LIN {X 0,Y 201.822,Z 772.403,A -85,B 0,C 180,E1 -21490.685,E2 -21490.685} C_VEL
LIN {X 0,Y 199.583,Z 777.598,A -85,B 0,C 180,E1 -21494.69,E2 -21494.69} C_VEL
LIN {X 0,Y 198.418,Z 780.58,A -85,B 0,C 180,E1 -21497.733,E2 -21497.733} C_VEL
LIN {X 0,Y 197.499,Z 783.514,A -85,B 0,C 180,E1 -21501.82,E2 -21501.82} C_VEL
LIN {X 0,Y 197.172,Z 785.274,A -85,B 0,C 180,E1 -21505.915,E2 -21505.915} C_VEL
LIN {X 0,Y 197.205,Z 785.884,A -85,B 0,C 180,E1 -21510.003,E2 -21510.003} C_VEL
LIN {X 0,Y 197.174,Z 785.308,A -85,B 0,C 180,E1 -21514.091,E2 -21514.091} C_VEL
LIN {X 0,Y 197.502,Z 783.592,A -85,B 0,C 180,E1 -21518.186,E2 -21518.186} C_VEL
LIN {X 0,Y 198.412,Z 780.698,A -85,B 0,C 180,E1 -21522.274,E2 -21522.274} C_VEL
LIN {X 0,Y 200.05,Z 776.56,A -85,B 0,C 180,E1 -21526.326,E2 -21526.326} C_VEL
LIN {X 0,Y 202.48,Z 770.918,A -85,B 0,C 180,E1 -21530.42,E2 -21530.42} C_VEL
LIN {X 0,Y 205.622,Z 764.102,A -85,B 0,C 180,E1 -21534.217,E2 -21534.217} C_VEL
LIN {X 0,Y 209.119,Z 756.621,A -85,B 0,C 180,E1 -21537.526,E2 -21537.526} C_VEL
LIN {X 0,Y 213.136,Z 748.003,A -85,B 0,C 180,E1 -21540.588,E2 -21540.588} C_VEL
LIN {X 0,Y 217.286,Z 738.403,A -85,B 0,C 180,E1 -21543.36,E2 -21543.36} C_VEL
LIN {X 0,Y 222.185,Z 726.543,A -85,B 0,C 180,E1 -21546.098,E2 -21546.098} C_VEL
LIN {X 0,Y 226.698,Z 714.44,A -85,B 0,C 180,E1 -21548.321,E2 -21548.321} C_VEL
LIN {X 0,Y 231.268,Z 700.736,A -85,B 0,C 180,E1 -21550.302,E2 -21550.302} C_VEL
LIN {X 0,Y 234.745,Z 688.105,A -85,B 0,C 180,E1 -21551.773,E2 -21551.773} C_VEL
LIN {X 0,Y 238.029,Z 673.847,A -85,B 0,C 180,E1 -21553.065,E2 -21553.065} C_VEL
LIN {X 0,Y 240.943,Z 658.425,A -85,B 0,C 180,E1 -21554.069,E2 -21554.069} C_VEL
LIN {X 0,Y 242.899,Z 642.997,A -85,B 0,C 180,E1 -21554.781,E2 -21554.781} C_VEL
LIN {X 0,Y 245.314,Z 607.777,A -85,B 0,C 180,E1 -21555.747,E2 -21555.747} C_VEL
LIN {X 0,Y 250.129,Z 529.748,A -85,B 0,C 180,E1 -21557.801,E2 -21557.801} C_VEL
LIN {X 0,Y 247.487,Z 500.103,A -85,B 0,C 180,E1 -21559.763,E2 -21559.763} C_VEL
LIN {X 0,Y 242.292,Z 488.929,A -85,B 0,C 180,E1 -21561.749,E2 -21561.749} C_VEL
LIN {X 0,Y 236.162,Z 477.144,A -85,B 0,C 180,E1 -21564.261,E2 -21564.261} C_VEL
LIN {X 0,Y 235.573,Z 475.998,A -85,B 0,C 180,E1 -21564.517,E2 -21564.517} C_VEL
LIN {X 0,Y 234.938,Z 476.527,A -85,B 0,C 180,E1 -21564.707,E2 -21564.707} C_VEL
LIN {X 0,Y 233.367,Z 478.417,A -85,B 0,C 180,E1 -21565.152,E2 -21565.152} C_VEL
LIN {X 0,Y 229.109,Z 492.899,A -85,B 0,C 180,E1 -21565.904,E2 -21565.904} C_VEL
LIN {X 0,Y 226.269,Z 500.58,A -85,B 0,C 180,E1 -21566.54,E2 -21566.54} C_VEL
LIN {X 0,Y 223.62,Z 505.401,A -85,B 0,C 180,E1 -21567.294,E2 -21567.294} C_VEL
LIN {X 0,Y 222.851,Z 506.93,A -85,B 0,C 180,E1 -21567.512,E2 -21567.512} C_VEL
LIN {X 0,Y 220.647,Z 514.522,A -85,B 0,C 180,E1 -21567.958,E2 -21567.958} C_VEL
LIN {X 0,Y 216.467,Z 529.632,A -85,B 0,C 180,E1 -21568.803,E2 -21568.803} C_VEL
LIN {X 0,Y 213.728,Z 537.354,A -85,B 0,C 180,E1 -21569.526,E2 -21569.526} C_VEL
LIN {X 0,Y 211.824,Z 540.819,A -85,B 0,C 180,E1 -21570.222,E2 -21570.222} C_VEL
LIN {X 0,Y 211.239,Z 542.496,A -85,B 0,C 180,E1 -21570.611,E2 -21570.611} C_VEL
LIN {X 0,Y 210.569,Z 548.908,A -85,B 0,C 180,E1 -21571.26,E2 -21571.26} C_VEL
LIN {X 0,Y 209.326,Z 568.525,A -85,B 0,C 180,E1 -21572.777,E2 -21572.777} C_VEL
LIN {X 0,Y 207.838,Z 584.724,A -85,B 0,C 180,E1 -21574.46,E2 -21574.46} C_VEL
LIN {X 0,Y 206.469,Z 599.243,A -85,B 0,C 180,E1 -21576.342,E2 -21576.342} C_VEL
LIN {X 0,Y 204.813,Z 613.408,A -85,B 0,C 180,E1 -21578.617,E2 -21578.617} C_VEL
LIN {X 0,Y 203.455,Z 626.182,A -85,B 0,C 180,E1 -21581.104,E2 -21581.104} C_VEL
LIN {X 0,Y 203.121,Z 628.887,A -85,B 0,C 180,E1 -21581.689,E2 -21581.689} C_VEL
LIN {X 0,Y 201.884,Z 633.396,A -85,B 0,C 180,E1 -21582.715,E2 -21582.715} C_VEL
LIN {X 0,Y 198.3,Z 640.449,A -85,B 0,C 180,E1 -21584.431,E2 -21584.431} C_VEL
LIN {X 0,Y 194.843,Z 647.157,A -85,B 0,C 180,E1 -21586.314,E2 -21586.314} C_VEL
LIN {X 0,Y 193.826,Z 651.128,A -85,B 0,C 180,E1 -21587.574,E2 -21587.574} C_VEL
LIN {X 0,Y 193.09,Z 661.092,A -85,B 0,C 180,E1 -21591.101,E2 -21591.101} C_VEL
LIN {X 0,Y 192.587,Z 669.692,A -85,B 0,C 180,E1 -21594.765,E2 -21594.765} C_VEL
LIN {X 0,Y 192.762,Z 677.727,A -85,B 0,C 180,E1 -21598.955,E2 -21598.955} C_VEL
LIN {X 0,Y 193.745,Z 684.126,A -85,B 0,C 180,E1 -21603.119,E2 -21603.119} C_VEL
LIN {X 0,Y 195.468,Z 689.048,A -85,B 0,C 180,E1 -21607.229,E2 -21607.229} C_VEL
LIN {X 0,Y 197.182,Z 691.828,A -85,B 0,C 180,E1 -21610.265,E2 -21610.265} C_VEL
LIN {X 0,Y 200.371,Z 694.455,A -85,B 0,C 180,E1 -21614.213,E2 -21614.213} C_VEL
LIN {X 0,Y 204.435,Z 695.846,A -85,B 0,C 180,E1 -21618.023,E2 -21618.023} C_VEL
LIN {X 0,Y 209.449,Z 696.032,A -85,B 0,C 180,E1 -21621.66,E2 -21621.66} C_VEL
LIN {X 0,Y 215.233,Z 695.074,A -85,B 0,C 180,E1 -21625.118,E2 -21625.118} C_VEL
LIN {X 0,Y 221.897,Z 692.933,A -85,B 0,C 180,E1 -21628.365,E2 -21628.365} C_VEL
LIN {X 0,Y 229.319,Z 689.599,A -85,B 0,C 180,E1 -21631.399,E2 -21631.399} C_VEL
LIN {X 0,Y 237.424,Z 685.083,A -85,B 0,C 180,E1 -21634.223,E2 -21634.223} C_VEL
LIN {X 0,Y 246.179,Z 679.309,A -85,B 0,C 180,E1 -21636.835,E2 -21636.835} C_VEL
LIN {X 0,Y 257.297,Z 670.804,A -85,B 0,C 180,E1 -21639.642,E2 -21639.642} C_VEL
LIN {X 0,Y 261.37,Z 667.332,A -85,B 0,C 180,E1 -21640.557,E2 -21640.557} C_VEL
LIN {X 0,Y 260.85,Z 668.132,A -85,B 0,C 180,E1 -21641.025,E2 -21641.025} C_VEL
LIN {X 0,Y 250.871,Z 678.551,A -85,B 0,C 180,E1 -21642.658,E2 -21642.658} C_VEL
LIN {X 0,Y 240.229,Z 688.929,A -85,B 0,C 180,E1 -21644.807,E2 -21644.807} C_VEL
LIN {X 0,Y 230.474,Z 697.908,A -85,B 0,C 180,E1 -21647.272,E2 -21647.272} C_VEL
LIN {X 0,Y 224.652,Z 703.275,A -85,B 0,C 180,E1 -21649.077,E2 -21649.077} C_VEL
LIN {X 0,Y 219.916,Z 716.568,A -85,B 0,C 180,E1 -21651.155,E2 -21651.155} C_VEL
LIN {X 0,Y 215.35,Z 728.239,A -85,B 0,C 180,E1 -21653.442,E2 -21653.442} C_VEL
LIN {X 0,Y 210.655,Z 738.922,A -85,B 0,C 180,E1 -21656.022,E2 -21656.022} C_VEL
LIN {X 0,Y 206.482,Z 748.241,A -85,B 0,C 180,E1 -21658.843,E2 -21658.843} C_VEL
LIN {X 0,Y 202.28,Z 756.832,A -85,B 0,C 180,E1 -21662.025,E2 -21662.025} C_VEL
LIN {X 0,Y 198.238,Z 765.11,A -85,B 0,C 180,E1 -21665.936,E2 -21665.936} C_VEL
LIN {X 0,Y 194.97,Z 771.854,A -85,B 0,C 180,E1 -21670.063,E2 -21670.063} C_VEL
LIN {X 0,Y 192.707,Z 776.915,A -85,B 0,C 180,E1 -21674.123,E2 -21674.123} C_VEL
LIN {X 0,Y 191.496,Z 779.895,A -85,B 0,C 180,E1 -21677.276,E2 -21677.276} C_VEL
LIN {X 0,Y 190.537,Z 782.809,A -85,B 0,C 180,E1 -21681.512,E2 -21681.512} C_VEL
LIN {X 0,Y 190.166,Z 784.542,A -85,B 0,C 180,E1 -21685.758,E2 -21685.758} C_VEL
LIN {X 0,Y 190.219,Z 785.129,A -85,B 0,C 180,E1 -21689.997,E2 -21689.997} C_VEL
LIN {X 0,Y 190.161,Z 784.528,A -85,B 0,C 180,E1 -21694.236,E2 -21694.236} C_VEL
LIN {X 0,Y 190.529,Z 782.778,A -85,B 0,C 180,E1 -21698.481,E2 -21698.481} C_VEL
LIN {X 0,Y 191.461,Z 779.852,A -85,B 0,C 180,E1 -21702.72,E2 -21702.72} C_VEL
LIN {X 0,Y 193.216,Z 775.677,A -85,B 0,C 180,E1 -21706.914,E2 -21706.914} C_VEL
LIN {X 0,Y 195.69,Z 770.141,A -85,B 0,C 180,E1 -21711.044,E2 -21711.044} C_VEL
LIN {X 0,Y 199.11,Z 763.093,A -85,B 0,C 180,E1 -21715.056,E2 -21715.056} C_VEL
LIN {X 0,Y 202.82,Z 755.539,A -85,B 0,C 180,E1 -21718.45,E2 -21718.45} C_VEL
LIN {X 0,Y 206.413,Z 748.128,A -85,B 0,C 180,E1 -21721.155,E2 -21721.155} C_VEL
LIN {X 0,Y 209.161,Z 741.992,A -85,B 0,C 180,E1 -21723.09,E2 -21723.09} C_VEL
LIN {X 0,Y 213.671,Z 731.872,A -85,B 0,C 180,E1 -21725.716,E2 -21725.716} C_VEL
LIN {X 0,Y 218.608,Z 719.81,A -85,B 0,C 180,E1 -21728.229,E2 -21728.229} C_VEL
LIN {X 0,Y 222.962,Z 707.693,A -85,B 0,C 180,E1 -21730.25,E2 -21730.25} C_VEL
LIN {X 0,Y 227.306,Z 693.77,A -85,B 0,C 180,E1 -21732.094,E2 -21732.094} C_VEL
LIN {X 0,Y 231.156,Z 678.884,A -85,B 0,C 180,E1 -21733.609,E2 -21733.609} C_VEL
LIN {X 0,Y 234.305,Z 663.775,A -85,B 0,C 180,E1 -21734.74,E2 -21734.74} C_VEL
LIN {X 0,Y 236.631,Z 648.765,A -85,B 0,C 180,E1 -21735.535,E2 -21735.535} C_VEL
LIN {X 0,Y 238.131,Z 633.231,A -85,B 0,C 180,E1 -21736.075,E2 -21736.075} C_VEL
LIN {X 0,Y 243.919,Z 543.137,A -85,B 0,C 180,E1 -21738.457,E2 -21738.457} C_VEL
LIN {X 0,Y 245.079,Z 524.954,A -85,B 0,C 180,E1 -21738.938,E2 -21738.938} C_VEL
LIN {X 0,Y 243.278,Z 494.459,A -85,B 0,C 180,E1 -21740.807,E2 -21740.807} C_VEL
LIN {X 0,Y 236.385,Z 475.168,A -85,B 0,C 180,E1 -21743.876,E2 -21743.876} C_VEL
LIN {X 0,Y 235.2,Z 472.841,A -85,B 0,C 180,E1 -21744.395,E2 -21744.395} C_VEL
LIN {X 0,Y 231.789,Z 467.9,A -85,B 0,C 180,E1 -21745.88,E2 -21745.88} C_VEL
LIN {X 0,Y 228.541,Z 461.545,A -85,B 0,C 180,E1 -21748.482,E2 -21748.482} C_VEL
LIN {X 0,Y 224.246,Z 454.408,A -85,B 0,C 180,E1 -21751.959,E2 -21751.959} C_VEL
LIN {X 0,Y 220.215,Z 447.535,A -85,B 0,C 180,E1 -21756.015,E2 -21756.015} C_VEL
LIN {X 0,Y 217.525,Z 443.267,A -85,B 0,C 180,E1 -21759.182,E2 -21759.182} C_VEL
LIN {X 0,Y 214.845,Z 439.385,A -85,B 0,C 180,E1 -21762.878,E2 -21762.878} C_VEL
LIN {X 0,Y 212.169,Z 434.902,A -85,B 0,C 180,E1 -21768.536,E2 -21768.536} C_VEL
LIN {X 0,Y 210.961,Z 433.332,A -85,B 0,C 180,E1 -21772.342,E2 -21772.342} C_VEL
LIN {X 0,Y 210.318,Z 432.552,A -85,B 0,C 180,E1 -21778.085,E2 -21778.085} C_VEL
LIN {X 0,Y 210.468,Z 432.967,A -85,B 0,C 180,E1 -21781.914,E2 -21781.914} C_VEL
LIN {X 0,Y 211.083,Z 434.259,A -85,B 0,C 180,E1 -21785.733,E2 -21785.733} C_VEL
LIN {X 0,Y 212.784,Z 438.249,A -85,B 0,C 180,E1 -21791.43,E2 -21791.43} C_VEL
LIN {X 0,Y 214.976,Z 442.904,A -85,B 0,C 180,E1 -21796.134,E2 -21796.134} C_VEL
LIN {X 0,Y 217.165,Z 447.743,A -85,B 0,C 180,E1 -21799.964,E2 -21799.964} C_VEL
LIN {X 0,Y 219.539,Z 453.313,A -85,B 0,C 180,E1 -21803.588,E2 -21803.588} C_VEL
LIN {X 0,Y 222.924,Z 461.584,A -85,B 0,C 180,E1 -21808.033,E2 -21808.033} C_VEL
LIN {X 0,Y 225.795,Z 469.875,A -85,B 0,C 180,E1 -21811.675,E2 -21811.675} C_VEL
LIN {X 0,Y 231.893,Z 480.479,A -85,B 0,C 180,E1 -21814.623,E2 -21814.623} C_VEL
LIN {X 0,Y 238.186,Z 492.808,A -85,B 0,C 180,E1 -21817.353,E2 -21817.353} C_VEL
LIN {X 0,Y 242.959,Z 503.436,A -85,B 0,C 180,E1 -21819.286,E2 -21819.286} C_VEL
LIN {X 0,Y 245.231,Z 531.174,A -85,B 0,C 180,E1 -21821.151,E2 -21821.151} C_VEL
LIN {X 0,Y 238.747,Z 630.862,A -85,B 0,C 180,E1 -21823.774,E2 -21823.774} C_VEL
LIN {X 0,Y 237.287,Z 647.272,A -85,B 0,C 180,E1 -21824.323,E2 -21824.323} C_VEL
LIN {X 0,Y 234.998,Z 662.794,A -85,B 0,C 180,E1 -21825.126,E2 -21825.126} C_VEL
LIN {X 0,Y 232.029,Z 677.096,A -85,B 0,C 180,E1 -21826.147,E2 -21826.147} C_VEL
LIN {X 0,Y 228.622,Z 690.646,A -85,B 0,C 180,E1 -21827.449,E2 -21827.449} C_VEL
LIN {X 0,Y 224.476,Z 704.619,A -85,B 0,C 180,E1 -21829.193,E2 -21829.193} C_VEL
LIN {X 0,Y 219.966,Z 717.307,A -85,B 0,C 180,E1 -21831.173,E2 -21831.173} C_VEL
LIN {X 0,Y 215.326,Z 728.928,A -85,B 0,C 180,E1 -21833.445,E2 -21833.445} C_VEL
LIN {X 0,Y 210.736,Z 739.581,A -85,B 0,C 180,E1 -21836.044,E2 -21836.044} C_VEL
LIN {X 0,Y 206.668,Z 748.771,A -85,B 0,C 180,E1 -21838.831,E2 -21838.831} C_VEL
LIN {X 0,Y 202.304,Z 757.469,A -85,B 0,C 180,E1 -21842.035,E2 -21842.035} C_VEL
LIN {X 0,Y 198.239,Z 765.746,A -85,B 0,C 180,E1 -21845.943,E2 -21845.943} C_VEL
LIN {X 0,Y 195.068,Z 772.389,A -85,B 0,C 180,E1 -21849.988,E2 -21849.988} C_VEL
LIN {X 0,Y 192.708,Z 777.584,A -85,B 0,C 180,E1 -21854.13,E2 -21854.13} C_VEL
LIN {X 0,Y 191.438,Z 780.566,A -85,B 0,C 180,E1 -21857.279,E2 -21857.279} C_VEL
LIN {X 0,Y 190.459,Z 783.5,A -85,B 0,C 180,E1 -21861.515,E2 -21861.515} C_VEL
LIN {X 0,Y 190.085,Z 785.261,A -85,B 0,C 180,E1 -21865.763,E2 -21865.763} C_VEL
LIN {X 0,Y 190.115,Z 785.87,A -85,B 0,C 180,E1 -21870.003,E2 -21870.003} C_VEL
LIN {X 0,Y 190.087,Z 785.294,A -85,B 0,C 180,E1 -21874.244,E2 -21874.244} C_VEL
LIN {X 0,Y 190.462,Z 783.577,A -85,B 0,C 180,E1 -21878.491,E2 -21878.491} C_VEL
LIN {X 0,Y 191.432,Z 780.683,A -85,B 0,C 180,E1 -21882.728,E2 -21882.728} C_VEL
LIN {X 0,Y 193.201,Z 776.544,A -85,B 0,C 180,E1 -21886.922,E2 -21886.922} C_VEL
LIN {X 0,Y 195.704,Z 771.063,A -85,B 0,C 180,E1 -21891.049,E2 -21891.049} C_VEL
LIN {X 0,Y 199.107,Z 764.084,A -85,B 0,C 180,E1 -21895.063,E2 -21895.063} C_VEL
LIN {X 0,Y 202.819,Z 756.602,A -85,B 0,C 180,E1 -21898.458,E2 -21898.458} C_VEL
LIN {X 0,Y 206.883,Z 748.24,A -85,B 0,C 180,E1 -21901.51,E2 -21901.51} C_VEL
LIN {X 0,Y 211.365,Z 738.381,A -85,B 0,C 180,E1 -21904.423,E2 -21904.423} C_VEL
LIN {X 0,Y 216.457,Z 726.518,A -85,B 0,C 180,E1 -21907.212,E2 -21907.212} C_VEL
LIN {X 0,Y 221.154,Z 714.412,A -85,B 0,C 180,E1 -21909.466,E2 -21909.466} C_VEL
LIN {X 0,Y 225.738,Z 701.182,A -85,B 0,C 180,E1 -21911.409,E2 -21911.409} C_VEL
LIN {X 0,Y 229.487,Z 688.066,A -85,B 0,C 180,E1 -21912.956,E2 -21912.956} C_VEL
LIN {X 0,Y 232.887,Z 673.799,A -85,B 0,C 180,E1 -21914.259,E2 -21914.259} C_VEL
LIN {X 0,Y 235.894,Z 658.359,A -85,B 0,C 180,E1 -21915.269,E2 -21915.269} C_VEL
LIN {X 0,Y 237.904,Z 642.891,A -85,B 0,C 180,E1 -21915.987,E2 -21915.987} C_VEL
LIN {X 0,Y 240.599,Z 605.269,A -85,B 0,C 180,E1 -21917.012,E2 -21917.012} C_VEL
LIN {X 0,Y 245.327,Z 530.521,A -85,B 0,C 180,E1 -21919.012,E2 -21919.012} C_VEL
LIN {X 0,Y 243.056,Z 503.406,A -85,B 0,C 180,E1 -21920.855,E2 -21920.855} C_VEL
LIN {X 0,Y 238.364,Z 493.238,A -85,B 0,C 180,E1 -21922.746,E2 -21922.746} C_VEL
LIN {X 0,Y 235.276,Z 487.003,A -85,B 0,C 180,E1 -21924.056,E2 -21924.056} C_VEL
LIN {X 0,Y 231.403,Z 499.009,A -85,B 0,C 180,E1 -21924.756,E2 -21924.756} C_VEL
LIN {X 0,Y 228.584,Z 505.786,A -85,B 0,C 180,E1 -21925.395,E2 -21925.395} C_VEL
LIN {X 0,Y 225.695,Z 510.994,A -85,B 0,C 180,E1 -21926.174,E2 -21926.174} C_VEL
LIN {X 0,Y 219.778,Z 531.993,A -85,B 0,C 180,E1 -21927.274,E2 -21927.274} C_VEL
LIN {X 0,Y 216.633,Z 540.683,A -85,B 0,C 180,E1 -21928.048,E2 -21928.048} C_VEL
LIN {X 0,Y 214.238,Z 545.202,A -85,B 0,C 180,E1 -21928.797,E2 -21928.797} C_VEL
LIN {X 0,Y 213.183,Z 546.946,A -85,B 0,C 180,E1 -21929.153,E2 -21929.153} C_VEL
LIN {X 0,Y 208.589,Z 562.229,A -85,B 0,C 180,E1 -21930.269,E2 -21930.269} C_VEL
LIN {X 0,Y 205.56,Z 570.357,A -85,B 0,C 180,E1 -21931.193,E2 -21931.193} C_VEL
LIN {X 0,Y 203.589,Z 574.003,A -85,B 0,C 180,E1 -21931.943,E2 -21931.943} C_VEL
LIN {X 0,Y 202.313,Z 575.787,A -85,B 0,C 180,E1 -21932.594,E2 -21932.594} C_VEL
LIN {X 0,Y 201.497,Z 579.228,A -85,B 0,C 180,E1 -21933.316,E2 -21933.316} C_VEL
LIN {X 0,Y 199.187,Z 601.55,A -85,B 0,C 180,E1 -21936.409,E2 -21936.409} C_VEL
LIN {X 0,Y 197.552,Z 615.998,A -85,B 0,C 180,E1 -21938.887,E2 -21938.887} C_VEL
LIN {X 0,Y 196.067,Z 628.546,A -85,B 0,C 180,E1 -21941.483,E2 -21941.483} C_VEL
LIN {X 0,Y 194.84,Z 639.997,A -85,B 0,C 180,E1 -21944.304,E2 -21944.304} C_VEL
LIN {X 0,Y 193.826,Z 651.128,A -85,B 0,C 180,E1 -21947.574,E2 -21947.574} C_VEL
LIN {X 0,Y 192.801,Z 655.036,A -85,B 0,C 180,E1 -21948.87,E2 -21948.87} C_VEL
LIN {X 0,Y 186.692,Z 665.347,A -85,B 0,C 180,E1 -21952.875,E2 -21952.875} C_VEL
LIN {X 0,Y 185.567,Z 668.609,A -85,B 0,C 180,E1 -21954.363,E2 -21954.363} C_VEL
LIN {X 0,Y 185.49,Z 669.682,A -85,B 0,C 180,E1 -21954.875,E2 -21954.875} C_VEL
LIN {X 0,Y 185.668,Z 677.422,A -85,B 0,C 180,E1 -21958.915,E2 -21958.915} C_VEL
LIN {X 0,Y 186.666,Z 684.138,A -85,B 0,C 180,E1 -21963.237,E2 -21963.237} C_VEL
LIN {X 0,Y 188.443,Z 689.389,A -85,B 0,C 180,E1 -21967.5,E2 -21967.5} C_VEL
LIN {X 0,Y 190.23,Z 692.476,A -85,B 0,C 180,E1 -21970.645,E2 -21970.645} C_VEL
LIN {X 0,Y 193.578,Z 695.43,A -85,B 0,C 180,E1 -21974.722,E2 -21974.722} C_VEL
LIN {X 0,Y 197.832,Z 697.169,A -85,B 0,C 180,E1 -21978.646,E2 -21978.646} C_VEL
LIN {X 0,Y 203.064,Z 697.7,A -85,B 0,C 180,E1 -21982.377,E2 -21982.377} C_VEL
LIN {X 0,Y 209.088,Z 697.103,A -85,B 0,C 180,E1 -21985.91,E2 -21985.91} C_VEL
LIN {X 0,Y 216.033,Z 695.352,A -85,B 0,C 180,E1 -21989.208,E2 -21989.208} C_VEL
LIN {X 0,Y 223.743,Z 692.456,A -85,B 0,C 180,E1 -21992.275,E2 -21992.275} C_VEL
LIN {X 0,Y 232.153,Z 688.406,A -85,B 0,C 180,E1 -21995.113,E2 -21995.113} C_VEL
LIN {X 0,Y 241.202,Z 683.173,A -85,B 0,C 180,E1 -21997.726,E2 -21997.726} C_VEL
LIN {X 0,Y 252,Z 675.891,A -85,B 0,C 180,E1 -22000.351,E2 -22000.351} C_VEL
LIN {X 0,Y 251.261,Z 676.688,A -85,B 0,C 180,E1 -22000.654,E2 -22000.654} C_VEL
LIN {X 0,Y 239.398,Z 687.495,A -85,B 0,C 180,E1 -22002.781,E2 -22002.781} C_VEL
LIN {X 0,Y 229.042,Z 696.348,A -85,B 0,C 180,E1 -22005.108,E2 -22005.108} C_VEL
LIN {X 0,Y 218.739,Z 704.998,A -85,B 0,C 180,E1 -22008.107,E2 -22008.107} C_VEL
LIN {X 0,Y 213.97,Z 717.756,A -85,B 0,C 180,E1 -22010.168,E2 -22010.168} C_VEL
LIN {X 0,Y 209.655,Z 728.263,A -85,B 0,C 180,E1 -22012.279,E2 -22012.279} C_VEL
LIN {X 0,Y 204.777,Z 738.944,A -85,B 0,C 180,E1 -22014.907,E2 -22014.907} C_VEL
LIN {X 0,Y 200.625,Z 747.724,A -85,B 0,C 180,E1 -22017.589,E2 -22017.589} C_VEL
LIN {X 0,Y 196.617,Z 755.678,A -85,B 0,C 180,E1 -22020.558,E2 -22020.558} C_VEL
LIN {X 0,Y 192.695,Z 763.212,A -85,B 0,C 180,E1 -22024.042,E2 -22024.042} C_VEL
LIN {X 0,Y 189.048,Z 770.233,A -85,B 0,C 180,E1 -22028.173,E2 -22028.173} C_VEL
LIN {X 0,Y 186.4,Z 775.746,A -85,B 0,C 180,E1 -22032.441,E2 -22032.441} C_VEL
LIN {X 0,Y 184.529,Z 779.91,A -85,B 0,C 180,E1 -22036.787,E2 -22036.787} C_VEL
LIN {X 0,Y 183.501,Z 782.823,A -85,B 0,C 180,E1 -22041.184,E2 -22041.184} C_VEL
LIN {X 0,Y 183.079,Z 784.556,A -85,B 0,C 180,E1 -22045.593,E2 -22045.593} C_VEL
LIN {X 0,Y 183.127,Z 785.142,A -85,B 0,C 180,E1 -22049.997,E2 -22049.997} C_VEL
LIN {X 0,Y 183.076,Z 784.542,A -85,B 0,C 180,E1 -22054.4,E2 -22054.4} C_VEL
LIN {X 0,Y 183.493,Z 782.792,A -85,B 0,C 180,E1 -22058.809,E2 -22058.809} C_VEL
LIN {X 0,Y 184.5,Z 779.865,A -85,B 0,C 180,E1 -22063.208,E2 -22063.208} C_VEL
LIN {X 0,Y 186.389,Z 775.691,A -85,B 0,C 180,E1 -22067.553,E2 -22067.553} C_VEL
LIN {X 0,Y 189.033,Z 770.155,A -85,B 0,C 180,E1 -22071.822,E2 -22071.822} C_VEL
LIN {X 0,Y 192.651,Z 763.107,A -85,B 0,C 180,E1 -22075.957,E2 -22075.957} C_VEL
LIN {X 0,Y 196.583,Z 755.554,A -85,B 0,C 180,E1 -22079.44,E2 -22079.44} C_VEL
LIN {X 0,Y 200.408,Z 747.899,A -85,B 0,C 180,E1 -22082.306,E2 -22082.306} C_VEL
LIN {X 0,Y 203.979,Z 740.396,A -85,B 0,C 180,E1 -22084.641,E2 -22084.641} C_VEL
LIN {X 0,Y 208.774,Z 730.004,A -85,B 0,C 180,E1 -22087.292,E2 -22087.292} C_VEL
LIN {X 0,Y 213.485,Z 718.691,A -85,B 0,C 180,E1 -22089.626,E2 -22089.626} C_VEL
LIN {X 0,Y 218.058,Z 706.38,A -85,B 0,C 180,E1 -22091.658,E2 -22091.658} C_VEL
LIN {X 0,Y 222.418,Z 692.669,A -85,B 0,C 180,E1 -22093.448,E2 -22093.448} C_VEL
LIN {X 0,Y 226.067,Z 678.917,A -85,B 0,C 180,E1 -22094.85,E2 -22094.85} C_VEL
LIN {X 0,Y 229.315,Z 663.818,A -85,B 0,C 180,E1 -22095.989,E2 -22095.989} C_VEL
LIN {X 0,Y 231.724,Z 648.828,A -85,B 0,C 180,E1 -22096.785,E2 -22096.785} C_VEL
LIN {X 0,Y 233.278,Z 633.332,A -85,B 0,C 180,E1 -22097.327,E2 -22097.327} C_VEL
LIN {X 0,Y 239.23,Z 544.075,A -85,B 0,C 180,E1 -22099.702,E2 -22099.702} C_VEL
LIN {X 0,Y 240.389,Z 524.977,A -85,B 0,C 180,E1 -22100.243,E2 -22100.243} C_VEL
LIN {X 0,Y 238.895,Z 497.387,A -85,B 0,C 180,E1 -22101.979,E2 -22101.979} C_VEL
LIN {X 0,Y 232.682,Z 479.464,A -85,B 0,C 180,E1 -22104.924,E2 -22104.924} C_VEL
LIN {X 0,Y 227.807,Z 472.074,A -85,B 0,C 180,E1 -22107.137,E2 -22107.137} C_VEL
LIN {X 0,Y 224.804,Z 467.654,A -85,B 0,C 180,E1 -22108.685,E2 -22108.685} C_VEL
LIN {X 0,Y 220.528,Z 460.091,A -85,B 0,C 180,E1 -22112.477,E2 -22112.477} C_VEL
LIN {X 0,Y 216.933,Z 453.901,A -85,B 0,C 180,E1 -22116.111,E2 -22116.111} C_VEL
LIN {X 0,Y 213.957,Z 449.133,A -85,B 0,C 180,E1 -22119.743,E2 -22119.743} C_VEL
LIN {X 0,Y 211.965,Z 446.122,A -85,B 0,C 180,E1 -22122.638,E2 -22122.638} C_VEL
LIN {X 0,Y 209.161,Z 441.496,A -85,B 0,C 180,E1 -22128.369,E2 -22128.369} C_VEL
LIN {X 0,Y 208.475,Z 440.425,A -85,B 0,C 180,E1 -22130.296,E2 -22130.296} C_VEL
LIN {X 0,Y 207.334,Z 439.366,A -85,B 0,C 180,E1 -22134.164,E2 -22134.164} C_VEL
LIN {X 0,Y 207.109,Z 438.88,A -85,B 0,C 180,E1 -22138.056,E2 -22138.056} C_VEL
LIN {X 0,Y 207.248,Z 439.318,A -85,B 0,C 180,E1 -22141.944,E2 -22141.944} C_VEL
LIN {X 0,Y 207.776,Z 440.659,A -85,B 0,C 180,E1 -22145.824,E2 -22145.824} C_VEL
LIN {X 0,Y 209.341,Z 444.672,A -85,B 0,C 180,E1 -22151.621,E2 -22151.621} C_VEL
LIN {X 0,Y 211.512,Z 449.47,A -85,B 0,C 180,E1 -22156.406,E2 -22156.406} C_VEL
LIN {X 0,Y 213.534,Z 454.252,A -85,B 0,C 180,E1 -22160.15,E2 -22160.15} C_VEL
LIN {X 0,Y 216.035,Z 460.411,A -85,B 0,C 180,E1 -22164.097,E2 -22164.097} C_VEL
LIN {X 0,Y 218.845,Z 467.738,A -85,B 0,C 180,E1 -22167.988,E2 -22167.988} C_VEL
LIN {X 0,Y 219.907,Z 470.403,A -85,B 0,C 180,E1 -22169.168,E2 -22169.168} C_VEL
LIN {X 0,Y 225.92,Z 480.721,A -85,B 0,C 180,E1 -22172.388,E2 -22172.388} C_VEL
LIN {X 0,Y 231.297,Z 490.851,A -85,B 0,C 180,E1 -22174.963,E2 -22174.963} C_VEL
LIN {X 0,Y 236,Z 500.733,A -85,B 0,C 180,E1 -22177.048,E2 -22177.048} C_VEL
LIN {X 0,Y 238.592,Z 506.663,A -85,B 0,C 180,E1 -22178.146,E2 -22178.146} C_VEL
LIN {X 0,Y 240.551,Z 532.006,A -85,B 0,C 180,E1 -22179.902,E2 -22179.902} C_VEL
LIN {X 0,Y 234.147,Z 627.191,A -85,B 0,C 180,E1 -22182.427,E2 -22182.427} C_VEL
LIN {X 0,Y 232.664,Z 645.062,A -85,B 0,C 180,E1 -22182.987,E2 -22182.987} C_VEL
LIN {X 0,Y 230.379,Z 660.554,A -85,B 0,C 180,E1 -22183.734,E2 -22183.734} C_VEL
LIN {X 0,Y 227.455,Z 674.873,A -85,B 0,C 180,E1 -22184.716,E2 -22184.716} C_VEL
LIN {X 0,Y 223.945,Z 688.894,A -85,B 0,C 180,E1 -22186.03,E2 -22186.03} C_VEL
LIN {X 0,Y 220.134,Z 701.678,A -85,B 0,C 180,E1 -22187.568,E2 -22187.568} C_VEL
LIN {X 0,Y 215.367,Z 714.979,A -85,B 0,C 180,E1 -22189.57,E2 -22189.57} C_VEL
LIN {X 0,Y 210.498,Z 726.987,A -85,B 0,C 180,E1 -22191.858,E2 -22191.858} C_VEL
LIN {X 0,Y 205.6,Z 737.956,A -85,B 0,C 180,E1 -22194.476,E2 -22194.476} C_VEL
LIN {X 0,Y 201.001,Z 747.846,A -85,B 0,C 180,E1 -22197.452,E2 -22197.452} C_VEL
LIN {X 0,Y 196.644,Z 756.272,A -85,B 0,C 180,E1 -22200.57,E2 -22200.57} C_VEL
LIN {X 0,Y 192.708,Z 763.807,A -85,B 0,C 180,E1 -22204.051,E2 -22204.051} C_VEL
LIN {X 0,Y 188.916,Z 771.231,A -85,B 0,C 180,E1 -22208.442,E2 -22208.442} C_VEL
LIN {X 0,Y 186.418,Z 776.376,A -85,B 0,C 180,E1 -22212.45,E2 -22212.45} C_VEL
LIN {X 0,Y 184.461,Z 780.553,A -85,B 0,C 180,E1 -22216.789,E2 -22216.789} C_VEL
LIN {X 0,Y 183.408,Z 783.486,A -85,B 0,C 180,E1 -22221.187,E2 -22221.187} C_VEL
LIN {X 0,Y 183.014,Z 785.247,A -85,B 0,C 180,E1 -22225.599,E2 -22225.599} C_VEL
LIN {X 0,Y 183.028,Z 785.856,A -85,B 0,C 180,E1 -22230.003,E2 -22230.003} C_VEL
LIN {X 0,Y 183.015,Z 785.28,A -85,B 0,C 180,E1 -22234.408,E2 -22234.408} C_VEL
LIN {X 0,Y 183.411,Z 783.563,A -85,B 0,C 180,E1 -22238.82,E2 -22238.82} C_VEL
LIN {X 0,Y 184.453,Z 780.668,A -85,B 0,C 180,E1 -22243.219,E2 -22243.219} C_VEL
LIN {X 0,Y 186.372,Z 776.529,A -85,B 0,C 180,E1 -22247.562,E2 -22247.562} C_VEL
LIN {X 0,Y 189.043,Z 771.046,A -85,B 0,C 180,E1 -22251.828,E2 -22251.828} C_VEL
LIN {X 0,Y 192.647,Z 764.066,A -85,B 0,C 180,E1 -22255.965,E2 -22255.965} C_VEL
LIN {X 0,Y 196.586,Z 756.583,A -85,B 0,C 180,E1 -22259.447,E2 -22259.447} C_VEL
LIN {X 0,Y 201.303,Z 747.153,A -85,B 0,C 180,E1 -22262.932,E2 -22262.932} C_VEL
LIN {X 0,Y 206.298,Z 736.664,A -85,B 0,C 180,E1 -22265.994,E2 -22265.994} C_VEL
LIN {X 0,Y 211.244,Z 725.454,A -85,B 0,C 180,E1 -22268.598,E2 -22268.598} C_VEL
LIN {X 0,Y 216.168,Z 713.135,A -85,B 0,C 180,E1 -22270.87,E2 -22270.87} C_VEL
LIN {X 0,Y 220.809,Z 699.918,A -85,B 0,C 180,E1 -22272.795,E2 -22272.795} C_VEL
LIN {X 0,Y 224.811,Z 686.156,A -85,B 0,C 180,E1 -22274.389,E2 -22274.389} C_VEL
LIN {X 0,Y 228.133,Z 672.581,A -85,B 0,C 180,E1 -22275.591,E2 -22275.591} C_VEL
LIN {X 0,Y 231.087,Z 657.44,A -85,B 0,C 180,E1 -22276.564,E2 -22276.564} C_VEL
LIN {X 0,Y 233.04,Z 642.784,A -85,B 0,C 180,E1 -22277.239,E2 -22277.239} C_VEL
LIN {X 0,Y 235.884,Z 604.057,A -85,B 0,C 180,E1 -22278.303,E2 -22278.303} C_VEL
LIN {X 0,Y 240.66,Z 532.179,A -85,B 0,C 180,E1 -22280.225,E2 -22280.225} C_VEL
LIN {X 0,Y 238.7,Z 506.724,A -85,B 0,C 180,E1 -22281.991,E2 -22281.991} C_VEL
LIN {X 0,Y 235.792,Z 500.201,A -85,B 0,C 180,E1 -22283.223,E2 -22283.223} C_VEL
LIN {X 0,Y 235.566,Z 500.122,A -85,B 0,C 180,E1 -22283.3,E2 -22283.3} C_VEL
LIN {X 0,Y 232.248,Z 508.399,A -85,B 0,C 180,E1 -22283.978,E2 -22283.978} C_VEL
LIN {X 0,Y 228.799,Z 514.787,A -85,B 0,C 180,E1 -22284.835,E2 -22284.835} C_VEL
LIN {X 0,Y 223.521,Z 533.48,A -85,B 0,C 180,E1 -22285.735,E2 -22285.735} C_VEL
LIN {X 0,Y 219.939,Z 543.423,A -85,B 0,C 180,E1 -22286.541,E2 -22286.541} C_VEL
LIN {X 0,Y 217.317,Z 548.651,A -85,B 0,C 180,E1 -22287.282,E2 -22287.282} C_VEL
LIN {X 0,Y 215.749,Z 551.434,A -85,B 0,C 180,E1 -22287.763,E2 -22287.763} C_VEL
LIN {X 0,Y 211.778,Z 564.569,A -85,B 0,C 180,E1 -22288.651,E2 -22288.651} C_VEL
LIN {X 0,Y 208.233,Z 573.872,A -85,B 0,C 180,E1 -22289.655,E2 -22289.655} C_VEL
LIN {X 0,Y 205.624,Z 578.752,A -85,B 0,C 180,E1 -22290.572,E2 -22290.572} C_VEL
LIN {X 0,Y 203.227,Z 582.177,A -85,B 0,C 180,E1 -22291.537,E2 -22291.537} C_VEL
LIN {X 0,Y 197.585,Z 596.555,A -85,B 0,C 180,E1 -22293.53,E2 -22293.53} C_VEL
LIN {X 0,Y 194.496,Z 602.76,A -85,B 0,C 180,E1 -22294.876,E2 -22294.876} C_VEL
LIN {X 0,Y 192.614,Z 605.229,A -85,B 0,C 180,E1 -22295.908,E2 -22295.908} C_VEL
LIN {X 0,Y 191.938,Z 606.321,A -85,B 0,C 180,E1 -22296.482,E2 -22296.482} C_VEL
LIN {X 0,Y 191.027,Z 610.771,A -85,B 0,C 180,E1 -22297.632,E2 -22297.632} C_VEL
LIN {X 0,Y 189.331,Z 625.927,A -85,B 0,C 180,E1 -22300.765,E2 -22300.765} C_VEL
LIN {X 0,Y 187.912,Z 638.083,A -85,B 0,C 180,E1 -22303.71,E2 -22303.71} C_VEL
LIN {X 0,Y 186.904,Z 649.205,A -85,B 0,C 180,E1 -22306.961,E2 -22306.961} C_VEL
LIN {X 0,Y 186.06,Z 660.07,A -85,B 0,C 180,E1 -22310.762,E2 -22310.762} C_VEL
LIN {X 0,Y 185.484,Z 669.037,A -85,B 0,C 180,E1 -22314.564,E2 -22314.564} C_VEL
LIN {X 0,Y 185.49,Z 669.682,A -85,B 0,C 180,E1 -22314.875,E2 -22314.875} C_VEL
LIN {X 0,Y 184.885,Z 672.807,A -85,B 0,C 180,E1 -22316.414,E2 -22316.414} C_VEL
LIN {X 0,Y 182.235,Z 677.532,A -85,B 0,C 180,E1 -22319,E2 -22319} C_VEL
LIN {X 0,Y 179.815,Z 681.818,A -85,B 0,C 180,E1 -22321.737,E2 -22321.737} C_VEL
LIN {X 0,Y 179.595,Z 684.222,A -85,B 0,C 180,E1 -22323.463,E2 -22323.463} C_VEL
LIN {X 0,Y 181.427,Z 689.679,A -85,B 0,C 180,E1 -22327.792,E2 -22327.792} C_VEL
LIN {X 0,Y 183.283,Z 692.951,A -85,B 0,C 180,E1 -22331.053,E2 -22331.053} C_VEL
LIN {X 0,Y 186.765,Z 696.244,A -85,B 0,C 180,E1 -22335.272,E2 -22335.272} C_VEL
LIN {X 0,Y 191.211,Z 698.336,A -85,B 0,C 180,E1 -22339.317,E2 -22339.317} C_VEL
LIN {X 0,Y 196.689,Z 699.244,A -85,B 0,C 180,E1 -22343.144,E2 -22343.144} C_VEL
LIN {X 0,Y 202.967,Z 699.048,A -85,B 0,C 180,E1 -22346.753,E2 -22346.753} C_VEL
LIN {X 0,Y 210.205,Z 697.711,A -85,B 0,C 180,E1 -22350.1,E2 -22350.1} C_VEL
LIN {X 0,Y 218.213,Z 695.261,A -85,B 0,C 180,E1 -22353.197,E2 -22353.197} C_VEL
LIN {X 0,Y 226.907,Z 691.685,A -85,B 0,C 180,E1 -22356.049,E2 -22356.049} C_VEL
LIN {X 0,Y 236.284,Z 686.953,A -85,B 0,C 180,E1 -22358.654,E2 -22358.654} C_VEL
LIN {X 0,Y 241.223,Z 684.131,A -85,B 0,C 180,E1 -22359.864,E2 -22359.864} C_VEL
LIN {X 0,Y 241.384,Z 684.28,A -85,B 0,C 180,E1 -22360.341,E2 -22360.341} C_VEL
LIN {X 0,Y 229.351,Z 693.906,A -85,B 0,C 180,E1 -22362.653,E2 -22362.653} C_VEL
LIN {X 0,Y 219.212,Z 701.537,A -85,B 0,C 180,E1 -22365.141,E2 -22365.141} C_VEL
LIN {X 0,Y 213.017,Z 706.39,A -85,B 0,C 180,E1 -22367.035,E2 -22367.035} C_VEL
LIN {X 0,Y 208.084,Z 718.945,A -85,B 0,C 180,E1 -22369.124,E2 -22369.124} C_VEL
LIN {X 0,Y 203.216,Z 730.221,A -85,B 0,C 180,E1 -22371.497,E2 -22371.497} C_VEL
LIN {X 0,Y 198.166,Z 740.58,A -85,B 0,C 180,E1 -22374.181,E2 -22374.181} C_VEL
LIN {X 0,Y 193.827,Z 749.352,A -85,B 0,C 180,E1 -22377.048,E2 -22377.048} C_VEL
LIN {X 0,Y 189.145,Z 757.977,A -85,B 0,C 180,E1 -22380.503,E2 -22380.503} C_VEL
LIN {X 0,Y 185.264,Z 765.144,A -85,B 0,C 180,E1 -22384.132,E2 -22384.132} C_VEL
LIN {X 0,Y 181.853,Z 771.286,A -85,B 0,C 180,E1 -22388.05,E2 -22388.05} C_VEL
LIN {X 0,Y 178.994,Z 776.946,A -85,B 0,C 180,E1 -22392.87,E2 -22392.87} C_VEL
LIN {X 0,Y 177.563,Z 779.925,A -85,B 0,C 180,E1 -22396.259,E2 -22396.259} C_VEL
LIN {X 0,Y 176.455,Z 782.838,A -85,B 0,C 180,E1 -22400.829,E2 -22400.829} C_VEL
LIN {X 0,Y 176.008,Z 784.57,A -85,B 0,C 180,E1 -22405.416,E2 -22405.416} C_VEL
LIN {X 0,Y 176.037,Z 785.156,A -85,B 0,C 180,E1 -22409.996,E2 -22409.996} C_VEL
LIN {X 0,Y 176.006,Z 784.556,A -85,B 0,C 180,E1 -22414.577,E2 -22414.577} C_VEL
LIN {X 0,Y 176.447,Z 782.806,A -85,B 0,C 180,E1 -22419.164,E2 -22419.164} C_VEL
LIN {X 0,Y 177.536,Z 779.879,A -85,B 0,C 180,E1 -22423.736,E2 -22423.736} C_VEL
LIN {X 0,Y 179.567,Z 775.705,A -85,B 0,C 180,E1 -22428.243,E2 -22428.243} C_VEL
LIN {X 0,Y 182.406,Z 770.169,A -85,B 0,C 180,E1 -22432.658,E2 -22432.658} C_VEL
LIN {X 0,Y 186.26,Z 763.122,A -85,B 0,C 180,E1 -22436.918,E2 -22436.918} C_VEL
LIN {X 0,Y 190.411,Z 755.569,A -85,B 0,C 180,E1 -22440.494,E2 -22440.494} C_VEL
LIN {X 0,Y 194.258,Z 748.17,A -85,B 0,C 180,E1 -22443.343,E2 -22443.343} C_VEL
LIN {X 0,Y 198.138,Z 740.413,A -85,B 0,C 180,E1 -22445.817,E2 -22445.817} C_VEL
LIN {X 0,Y 203.144,Z 730.022,A -85,B 0,C 180,E1 -22448.511,E2 -22448.511} C_VEL
LIN {X 0,Y 208.055,Z 718.711,A -85,B 0,C 180,E1 -22450.875,E2 -22450.875} C_VEL
LIN {X 0,Y 212.798,Z 706.402,A -85,B 0,C 180,E1 -22452.931,E2 -22452.931} C_VEL
LIN {X 0,Y 217.125,Z 693.364,A -85,B 0,C 180,E1 -22454.66,E2 -22454.66} C_VEL
LIN {X 0,Y 221.094,Z 678.949,A -85,B 0,C 180,E1 -22456.147,E2 -22456.147} C_VEL
LIN {X 0,Y 224.454,Z 663.86,A -85,B 0,C 180,E1 -22457.289,E2 -22457.289} C_VEL
LIN {X 0,Y 226.932,Z 648.889,A -85,B 0,C 180,E1 -22458.089,E2 -22458.089} C_VEL
LIN {X 0,Y 228.539,Z 633.431,A -85,B 0,C 180,E1 -22458.632,E2 -22458.632} C_VEL
LIN {X 0,Y 234.76,Z 543.311,A -85,B 0,C 180,E1 -22461.048,E2 -22461.048} C_VEL
LIN {X 0,Y 235.864,Z 526.059,A -85,B 0,C 180,E1 -22461.536,E2 -22461.536} C_VEL
LIN {X 0,Y 234.618,Z 500.314,A -85,B 0,C 180,E1 -22463.195,E2 -22463.195} C_VEL
LIN {X 0,Y 229.22,Z 484.16,A -85,B 0,C 180,E1 -22465.923,E2 -22465.923} C_VEL
LIN {X 0,Y 222.035,Z 473.504,A -85,B 0,C 180,E1 -22469.442,E2 -22469.442} C_VEL
LIN {X 0,Y 217.838,Z 467.78,A -85,B 0,C 180,E1 -22471.846,E2 -22471.846} C_VEL
LIN {X 0,Y 214.044,Z 461.086,A -85,B 0,C 180,E1 -22475.768,E2 -22475.768} C_VEL
LIN {X 0,Y 210.984,Z 455.871,A -85,B 0,C 180,E1 -22479.527,E2 -22479.527} C_VEL
LIN {X 0,Y 207.847,Z 451.149,A -85,B 0,C 180,E1 -22484.306,E2 -22484.306} C_VEL
LIN {X 0,Y 206.147,Z 448.082,A -85,B 0,C 180,E1 -22488.197,E2 -22488.197} C_VEL
LIN {X 0,Y 205.479,Z 446.955,A -85,B 0,C 180,E1 -22490.153,E2 -22490.153} C_VEL
LIN {X 0,Y 204.871,Z 446.193,A -85,B 0,C 180,E1 -22492.113,E2 -22492.113} C_VEL
LIN {X 0,Y 203.905,Z 445.199,A -85,B 0,C 180,E1 -22498.147,E2 -22498.147} C_VEL
LIN {X 0,Y 204.034,Z 445.656,A -85,B 0,C 180,E1 -22501.974,E2 -22501.974} C_VEL
LIN {X 0,Y 204.54,Z 447.071,A -85,B 0,C 180,E1 -22505.917,E2 -22505.917} C_VEL
LIN {X 0,Y 206.006,Z 451.201,A -85,B 0,C 180,E1 -22511.812,E2 -22511.812} C_VEL
LIN {X 0,Y 208.044,Z 456.043,A -85,B 0,C 180,E1 -22516.687,E2 -22516.687} C_VEL
LIN {X 0,Y 210,Z 460.953,A -85,B 0,C 180,E1 -22520.446,E2 -22520.446} C_VEL
LIN {X 0,Y 211.862,Z 465.675,A -85,B 0,C 180,E1 -22523.458,E2 -22523.458} C_VEL
LIN {X 0,Y 213.605,Z 470.187,A -85,B 0,C 180,E1 -22525.977,E2 -22525.977} C_VEL
LIN {X 0,Y 218.427,Z 478.171,A -85,B 0,C 180,E1 -22528.989,E2 -22528.989} C_VEL
LIN {X 0,Y 223.698,Z 487.608,A -85,B 0,C 180,E1 -22531.895,E2 -22531.895} C_VEL
LIN {X 0,Y 228.895,Z 497.846,A -85,B 0,C 180,E1 -22534.478,E2 -22534.478} C_VEL
LIN {X 0,Y 233.309,Z 507.607,A -85,B 0,C 180,E1 -22536.517,E2 -22536.517} C_VEL
LIN {X 0,Y 234.371,Z 510.608,A -85,B 0,C 180,E1 -22537.014,E2 -22537.014} C_VEL
LIN {X 0,Y 235.983,Z 533.03,A -85,B 0,C 180,E1 -22538.611,E2 -22538.611} C_VEL
LIN {X 0,Y 229.412,Z 627.09,A -85,B 0,C 180,E1 -22541.117,E2 -22541.117} C_VEL
LIN {X 0,Y 227.892,Z 644.999,A -85,B 0,C 180,E1 -22541.684,E2 -22541.684} C_VEL
LIN {X 0,Y 225.525,Z 660.511,A -85,B 0,C 180,E1 -22542.429,E2 -22542.429} C_VEL
LIN {X 0,Y 222.518,Z 674.84,A -85,B 0,C 180,E1 -22543.417,E2 -22543.417} C_VEL
LIN {X 0,Y 218.887,Z 688.867,A -85,B 0,C 180,E1 -22544.738,E2 -22544.738} C_VEL
LIN {X 0,Y 214.846,Z 701.871,A -85,B 0,C 180,E1 -22546.315,E2 -22546.315} C_VEL
LIN {X 0,Y 210.002,Z 714.958,A -85,B 0,C 180,E1 -22548.311,E2 -22548.311} C_VEL
LIN {X 0,Y 204.922,Z 726.968,A -85,B 0,C 180,E1 -22550.623,E2 -22550.623} C_VEL
LIN {X 0,Y 199.832,Z 737.939,A -85,B 0,C 180,E1 -22553.286,E2 -22553.286} C_VEL
LIN {X 0,Y 195.458,Z 746.73,A -85,B 0,C 180,E1 -22555.942,E2 -22555.942} C_VEL
LIN {X 0,Y 191.164,Z 755.04,A -85,B 0,C 180,E1 -22559.027,E2 -22559.027} C_VEL
LIN {X 0,Y 187.406,Z 761.797,A -85,B 0,C 180,E1 -22562.05,E2 -22562.05} C_VEL
LIN {X 0,Y 183.345,Z 769.23,A -85,B 0,C 180,E1 -22566.27,E2 -22566.27} C_VEL
LIN {X 0,Y 180.211,Z 775.131,A -85,B 0,C 180,E1 -22570.645,E2 -22570.645} C_VEL
LIN {X 0,Y 178.434,Z 778.612,A -85,B 0,C 180,E1 -22574,E2 -22574} C_VEL
LIN {X 0,Y 176.86,Z 782.156,A -85,B 0,C 180,E1 -22578.543,E2 -22578.543} C_VEL
LIN {X 0,Y 176.072,Z 784.497,A -85,B 0,C 180,E1 -22583.126,E2 -22583.126} C_VEL
LIN {X 0,Y 175.887,Z 785.685,A -85,B 0,C 180,E1 -22587.714,E2 -22587.714} C_VEL
LIN {X 0,Y 175.937,Z 785.842,A -85,B 0,C 180,E1 -22590.004,E2 -22590.004} C_VEL
LIN {X 0,Y 175.937,Z 785.266,A -85,B 0,C 180,E1 -22594.586,E2 -22594.586} C_VEL
LIN {X 0,Y 176.357,Z 783.548,A -85,B 0,C 180,E1 -22599.176,E2 -22599.176} C_VEL
LIN {X 0,Y 177.492,Z 780.653,A -85,B 0,C 180,E1 -22603.747,E2 -22603.747} C_VEL
LIN {X 0,Y 179.551,Z 776.513,A -85,B 0,C 180,E1 -22608.252,E2 -22608.252} C_VEL
LIN {X 0,Y 182.415,Z 771.029,A -85,B 0,C 180,E1 -22612.664,E2 -22612.664} C_VEL
LIN {X 0,Y 186.244,Z 764.048,A -85,B 0,C 180,E1 -22616.928,E2 -22616.928} C_VEL
LIN {X 0,Y 190.413,Z 756.564,A -85,B 0,C 180,E1 -22620.501,E2 -22620.501} C_VEL
LIN {X 0,Y 195.041,Z 747.73,A -85,B 0,C 180,E1 -22623.877,E2 -22623.877} C_VEL
LIN {X 0,Y 199.744,Z 738.337,A -85,B 0,C 180,E1 -22626.74,E2 -22626.74} C_VEL
LIN {X 0,Y 205.272,Z 726.468,A -85,B 0,C 180,E1 -22629.622,E2 -22629.622} C_VEL
LIN {X 0,Y 210.359,Z 714.355,A -85,B 0,C 180,E1 -22631.931,E2 -22631.931} C_VEL
LIN {X 0,Y 215.369,Z 700.737,A -85,B 0,C 180,E1 -22633.971,E2 -22633.971} C_VEL
LIN {X 0,Y 219.276,Z 687.989,A -85,B 0,C 180,E1 -22635.494,E2 -22635.494} C_VEL
LIN {X 0,Y 222.954,Z 673.704,A -85,B 0,C 180,E1 -22636.802,E2 -22636.802} C_VEL
LIN {X 0,Y 226.129,Z 658.224,A -85,B 0,C 180,E1 -22637.825,E2 -22637.825} C_VEL
LIN {X 0,Y 228.288,Z 642.674,A -85,B 0,C 180,E1 -22638.545,E2 -22638.545} C_VEL
LIN {X 0,Y 231.375,Z 601.832,A -85,B 0,C 180,E1 -22639.67,E2 -22639.67} C_VEL
LIN {X 0,Y 236.079,Z 532.786,A -85,B 0,C 180,E1 -22641.543,E2 -22641.543} C_VEL
LIN {X 0,Y 234.712,Z 513.636,A -85,B 0,C 180,E1 -22642.903,E2 -22642.903} C_VEL
LIN {X 0,Y 232.224,Z 518.14,A -85,B 0,C 180,E1 -22643.488,E2 -22643.488} C_VEL
LIN {X 0,Y 227.045,Z 536.113,A -85,B 0,C 180,E1 -22644.318,E2 -22644.318} C_VEL
LIN {X 0,Y 223.137,Z 546.732,A -85,B 0,C 180,E1 -22645.143,E2 -22645.143} C_VEL
LIN {X 0,Y 220.154,Z 552.683,A -85,B 0,C 180,E1 -22645.927,E2 -22645.927} C_VEL
LIN {X 0,Y 218.758,Z 555.05,A -85,B 0,C 180,E1 -22646.331,E2 -22646.331} C_VEL
LIN {X 0,Y 215.132,Z 566.893,A -85,B 0,C 180,E1 -22647.083,E2 -22647.083} C_VEL
LIN {X 0,Y 211.2,Z 577.097,A -85,B 0,C 180,E1 -22648.112,E2 -22648.112} C_VEL
LIN {X 0,Y 208.187,Z 582.886,A -85,B 0,C 180,E1 -22649.08,E2 -22649.08} C_VEL
LIN {X 0,Y 205.139,Z 587.369,A -85,B 0,C 180,E1 -22650.214,E2 -22650.214} C_VEL
LIN {X 0,Y 200.166,Z 599.812,A -85,B 0,C 180,E1 -22651.848,E2 -22651.848} C_VEL
LIN {X 0,Y 196.5,Z 607.159,A -85,B 0,C 180,E1 -22653.314,E2 -22653.314} C_VEL
LIN {X 0,Y 194.285,Z 610.352,A -85,B 0,C 180,E1 -22654.367,E2 -22654.367} C_VEL
LIN {X 0,Y 192.499,Z 612.331,A -85,B 0,C 180,E1 -22655.318,E2 -22655.318} C_VEL
LIN {X 0,Y 186.488,Z 625.463,A -85,B 0,C 180,E1 -22658.297,E2 -22658.297} C_VEL
LIN {X 0,Y 183.527,Z 630.744,A -85,B 0,C 180,E1 -22660.131,E2 -22660.131} C_VEL
LIN {X 0,Y 182.205,Z 632.403,A -85,B 0,C 180,E1 -22661.153,E2 -22661.153} C_VEL
LIN {X 0,Y 181.549,Z 633.474,A -85,B 0,C 180,E1 -22661.959,E2 -22661.959} C_VEL
LIN {X 0,Y 180.915,Z 637.21,A -85,B 0,C 180,E1 -22663.351,E2 -22663.351} C_VEL
LIN {X 0,Y 179.642,Z 650.993,A -85,B 0,C 180,E1 -22667.575,E2 -22667.575} C_VEL
LIN {X 0,Y 178.786,Z 661.709,A -85,B 0,C 180,E1 -22671.523,E2 -22671.523} C_VEL
LIN {X 0,Y 178.419,Z 670.59,A -85,B 0,C 180,E1 -22675.481,E2 -22675.481} C_VEL
LIN {X 0,Y 178.579,Z 676.984,A -85,B 0,C 180,E1 -22678.872,E2 -22678.872} C_VEL
LIN {X 0,Y 179.595,Z 684.222,A -85,B 0,C 180,E1 -22683.463,E2 -22683.463} C_VEL
LIN {X 0,Y 179.518,Z 686.533,A -85,B 0,C 180,E1 -22685.205,E2 -22685.205} C_VEL
LIN {X 0,Y 177.938,Z 689.968,A -85,B 0,C 180,E1 -22688.145,E2 -22688.145} C_VEL
LIN {X 0,Y 176.873,Z 692.452,A -85,B 0,C 180,E1 -22690.563,E2 -22690.563} C_VEL
LIN {X 0,Y 177.066,Z 694.185,A -85,B 0,C 180,E1 -22692.397,E2 -22692.397} C_VEL
LIN {X 0,Y 177.431,Z 694.715,A -85,B 0,C 180,E1 -22692.999,E2 -22692.999} C_VEL
LIN {X 0,Y 179.973,Z 697.013,A -85,B 0,C 180,E1 -22695.864,E2 -22695.864} C_VEL
LIN {X 0,Y 184.615,Z 699.449,A -85,B 0,C 180,E1 -22700.036,E2 -22700.036} C_VEL
LIN {X 0,Y 190.332,Z 700.707,A -85,B 0,C 180,E1 -22703.964,E2 -22703.964} C_VEL
LIN {X 0,Y 196.869,Z 700.876,A -85,B 0,C 180,E1 -22707.651,E2 -22707.651} C_VEL
LIN {X 0,Y 204.4,Z 699.922,A -85,B 0,C 180,E1 -22711.048,E2 -22711.048} C_VEL
LIN {X 0,Y 212.692,Z 697.903,A -85,B 0,C 180,E1 -22714.175,E2 -22714.175} C_VEL
LIN {X 0,Y 221.688,Z 694.799,A -85,B 0,C 180,E1 -22717.037,E2 -22717.037} C_VEL
LIN {X 0,Y 231.363,Z 690.589,A -85,B 0,C 180,E1 -22719.636,E2 -22719.636} C_VEL
LIN {X 0,Y 230.224,Z 691.657,A -85,B 0,C 180,E1 -22720.252,E2 -22720.252} C_VEL
LIN {X 0,Y 219.397,Z 699.228,A -85,B 0,C 180,E1 -22722.54,E2 -22722.54} C_VEL
LIN {X 0,Y 207.48,Z 707.443,A -85,B 0,C 180,E1 -22725.848,E2 -22725.848} C_VEL
LIN {X 0,Y 202.28,Z 720.091,A -85,B 0,C 180,E1 -22728.02,E2 -22728.02} C_VEL
LIN {X 0,Y 196.791,Z 732.113,A -85,B 0,C 180,E1 -22730.658,E2 -22730.658} C_VEL
LIN {X 0,Y 191.614,Z 742.206,A -85,B 0,C 180,E1 -22733.411,E2 -22733.411} C_VEL
LIN {X 0,Y 186.446,Z 752.045,A -85,B 0,C 180,E1 -22736.864,E2 -22736.864} C_VEL
LIN {X 0,Y 181.712,Z 760.213,A -85,B 0,C 180,E1 -22740.45,E2 -22740.45} C_VEL
LIN {X 0,Y 177.773,Z 766.957,A -85,B 0,C 180,E1 -22744.22,E2 -22744.22} C_VEL
LIN {X 0,Y 174.198,Z 773.199,A -85,B 0,C 180,E1 -22748.706,E2 -22748.706} C_VEL
LIN {X 0,Y 171.593,Z 778.02,A -85,B 0,C 180,E1 -22753.336,E2 -22753.336} C_VEL
LIN {X 0,Y 169.941,Z 781.548,A -85,B 0,C 180,E1 -22758.063,E2 -22758.063} C_VEL
LIN {X 0,Y 169.096,Z 783.862,A -85,B 0,C 180,E1 -22762.834,E2 -22762.834} C_VEL
LIN {X 0,Y 168.887,Z 785.02,A -85,B 0,C 180,E1 -22767.611,E2 -22767.611} C_VEL
LIN {X 0,Y 168.949,Z 785.17,A -85,B 0,C 180,E1 -22769.996,E2 -22769.996} C_VEL
LIN {X 0,Y 168.929,Z 784.569,A -85,B 0,C 180,E1 -22774.769,E2 -22774.769} C_VEL
LIN {X 0,Y 169.398,Z 782.819,A -85,B 0,C 180,E1 -22779.549,E2 -22779.549} C_VEL
LIN {X 0,Y 170.592,Z 779.893,A -85,B 0,C 180,E1 -22784.307,E2 -22784.307} C_VEL
LIN {X 0,Y 172.762,Z 775.719,A -85,B 0,C 180,E1 -22788.988,E2 -22788.988} C_VEL
LIN {X 0,Y 175.815,Z 770.183,A -85,B 0,C 180,E1 -22793.558,E2 -22793.558} C_VEL
LIN {X 0,Y 179.899,Z 763.137,A -85,B 0,C 180,E1 -22797.952,E2 -22797.952} C_VEL
LIN {X 0,Y 184.303,Z 755.584,A -85,B 0,C 180,E1 -22801.619,E2 -22801.619} C_VEL
LIN {X 0,Y 188.559,Z 747.676,A -85,B 0,C 180,E1 -22804.736,E2 -22804.736} C_VEL
LIN {X 0,Y 194.087,Z 737.2,A -85,B 0,C 180,E1 -22807.989,E2 -22807.989} C_VEL
LIN {X 0,Y 199.862,Z 725.165,A -85,B 0,C 180,E1 -22810.91,E2 -22810.91} C_VEL
LIN {X 0,Y 205.159,Z 712.871,A -85,B 0,C 180,E1 -22813.241,E2 -22813.241} C_VEL
LIN {X 0,Y 210.206,Z 699.237,A -85,B 0,C 180,E1 -22815.274,E2 -22815.274} C_VEL
LIN {X 0,Y 214.349,Z 685.892,A -85,B 0,C 180,E1 -22816.841,E2 -22816.841} C_VEL
LIN {X 0,Y 218.175,Z 671.059,A -85,B 0,C 180,E1 -22818.147,E2 -22818.147} C_VEL
LIN {X 0,Y 221.146,Z 656.258,A -85,B 0,C 180,E1 -22819.087,E2 -22819.087} C_VEL
LIN {X 0,Y 223.232,Z 640.928,A -85,B 0,C 180,E1 -22819.765,E2 -22819.765} C_VEL
LIN {X 0,Y 229.59,Z 554.603,A -85,B 0,C 180,E1 -22822.112,E2 -22822.112} C_VEL
LIN {X 0,Y 231.477,Z 527.541,A -85,B 0,C 180,E1 -22822.856,E2 -22822.856} C_VEL
LIN {X 0,Y 230.457,Z 503.248,A -85,B 0,C 180,E1 -22824.452,E2 -22824.452} C_VEL
LIN {X 0,Y 225.899,Z 489.235,A -85,B 0,C 180,E1 -22826.903,E2 -22826.903} C_VEL
LIN {X 0,Y 219.6,Z 479.595,A -85,B 0,C 180,E1 -22830.145,E2 -22830.145} C_VEL
LIN {X 0,Y 213.836,Z 471.887,A -85,B 0,C 180,E1 -22833.537,E2 -22833.537} C_VEL
LIN {X 0,Y 211.097,Z 468.196,A -85,B 0,C 180,E1 -22835.408,E2 -22835.408} C_VEL
LIN {X 0,Y 208.01,Z 462.78,A -85,B 0,C 180,E1 -22839.221,E2 -22839.221} C_VEL
LIN {X 0,Y 206.009,Z 459.587,A -85,B 0,C 180,E1 -22842.12,E2 -22842.12} C_VEL
LIN {X 0,Y 203.04,Z 454.646,A -85,B 0,C 180,E1 -22848.014,E2 -22848.014} C_VEL
LIN {X 0,Y 202.333,Z 453.43,A -85,B 0,C 180,E1 -22849.999,E2 -22849.999} C_VEL
LIN {X 0,Y 201.718,Z 452.603,A -85,B 0,C 180,E1 -22851.989,E2 -22851.989} C_VEL
LIN {X 0,Y 200.768,Z 451.594,A -85,B 0,C 180,E1 -22857.994,E2 -22857.994} C_VEL
LIN {X 0,Y 200.772,Z 451.977,A -85,B 0,C 180,E1 -22862.006,E2 -22862.006} C_VEL
LIN {X 0,Y 201.162,Z 453.436,A -85,B 0,C 180,E1 -22866.016,E2 -22866.016} C_VEL
LIN {X 0,Y 201.945,Z 456.076,A -85,B 0,C 180,E1 -22870.021,E2 -22870.021} C_VEL
LIN {X 0,Y 203.723,Z 460.54,A -85,B 0,C 180,E1 -22875.012,E2 -22875.012} C_VEL
LIN {X 0,Y 205.114,Z 463.927,A -85,B 0,C 180,E1 -22877.961,E2 -22877.961} C_VEL
LIN {X 0,Y 207.348,Z 469.873,A -85,B 0,C 180,E1 -22882.153,E2 -22882.153} C_VEL
LIN {X 0,Y 212.273,Z 477.815,A -85,B 0,C 180,E1 -22885.823,E2 -22885.823} C_VEL
LIN {X 0,Y 216.169,Z 484.488,A -85,B 0,C 180,E1 -22888.331,E2 -22888.331} C_VEL
LIN {X 0,Y 221.997,Z 495.388,A -85,B 0,C 180,E1 -22891.657,E2 -22891.657} C_VEL
LIN {X 0,Y 227.021,Z 505.916,A -85,B 0,C 180,E1 -22894.233,E2 -22894.233} C_VEL
LIN {X 0,Y 230.2,Z 513.508,A -85,B 0,C 180,E1 -22895.772,E2 -22895.772} C_VEL
LIN {X 0,Y 231.487,Z 534.891,A -85,B 0,C 180,E1 -22897.295,E2 -22897.295} C_VEL
LIN {X 0,Y 224.422,Z 632.342,A -85,B 0,C 180,E1 -22899.898,E2 -22899.898} C_VEL
LIN {X 0,Y 222.81,Z 648.164,A -85,B 0,C 180,E1 -22900.456,E2 -22900.456} C_VEL
LIN {X 0,Y 220.254,Z 663.4,A -85,B 0,C 180,E1 -22901.254,E2 -22901.254} C_VEL
LIN {X 0,Y 216.881,Z 678.094,A -85,B 0,C 180,E1 -22902.339,E2 -22902.339} C_VEL
LIN {X 0,Y 213.033,Z 691.742,A -85,B 0,C 180,E1 -22903.705,E2 -22903.705} C_VEL
LIN {X 0,Y 208.766,Z 704.551,A -85,B 0,C 180,E1 -22905.357,E2 -22905.357} C_VEL
LIN {X 0,Y 203.759,Z 717.248,A -85,B 0,C 180,E1 -22907.403,E2 -22907.403} C_VEL
LIN {X 0,Y 198.551,Z 728.874,A -85,B 0,C 180,E1 -22909.765,E2 -22909.765} C_VEL
LIN {X 0,Y 193.317,Z 739.531,A -85,B 0,C 180,E1 -22912.492,E2 -22912.492} C_VEL
LIN {X 0,Y 188.613,Z 748.661,A -85,B 0,C 180,E1 -22915.421,E2 -22915.421} C_VEL
LIN {X 0,Y 183.647,Z 757.424,A -85,B 0,C 180,E1 -22918.898,E2 -22918.898} C_VEL
LIN {X 0,Y 178.847,Z 765.703,A -85,B 0,C 180,E1 -22923.138,E2 -22923.138} C_VEL
LIN {X 0,Y 175.298,Z 771.914,A -85,B 0,C 180,E1 -22927.237,E2 -22927.237} C_VEL
LIN {X 0,Y 172.176,Z 777.543,A -85,B 0,C 180,E1 -22932.177,E2 -22932.177} C_VEL
LIN {X 0,Y 170.56,Z 780.525,A -85,B 0,C 180,E1 -22935.69,E2 -22935.69} C_VEL
LIN {X 0,Y 169.323,Z 783.459,A -85,B 0,C 180,E1 -22940.447,E2 -22940.447} C_VEL
LIN {X 0,Y 168.852,Z 785.219,A -85,B 0,C 180,E1 -22945.229,E2 -22945.229} C_VEL
LIN {X 0,Y 168.85,Z 785.829,A -85,B 0,C 180,E1 -22950.004,E2 -22950.004} C_VEL
LIN {X 0,Y 168.854,Z 785.252,A -85,B 0,C 180,E1 -22954.779,E2 -22954.779} C_VEL
LIN {X 0,Y 169.325,Z 783.534,A -85,B 0,C 180,E1 -22959.56,E2 -22959.56} C_VEL
LIN {X 0,Y 170.55,Z 780.638,A -85,B 0,C 180,E1 -22964.318,E2 -22964.318} C_VEL
LIN {X 0,Y 172.748,Z 776.497,A -85,B 0,C 180,E1 -22968.997,E2 -22968.997} C_VEL
LIN {X 0,Y 175.824,Z 771.013,A -85,B 0,C 180,E1 -22973.564,E2 -22973.564} C_VEL
LIN {X 0,Y 179.872,Z 764.03,A -85,B 0,C 180,E1 -22977.964,E2 -22977.964} C_VEL
LIN {X 0,Y 184.299,Z 756.545,A -85,B 0,C 180,E1 -22981.627,E2 -22981.627} C_VEL
LIN {X 0,Y 189.565,Z 746.911,A -85,B 0,C 180,E1 -22985.35,E2 -22985.35} C_VEL
LIN {X 0,Y 194.942,Z 736.618,A -85,B 0,C 180,E1 -22988.458,E2 -22988.458} C_VEL
LIN {X 0,Y 200.303,Z 725.402,A -85,B 0,C 180,E1 -22991.142,E2 -22991.142} C_VEL
LIN {X 0,Y 205.631,Z 713.077,A -85,B 0,C 180,E1 -22993.462,E2 -22993.462} C_VEL
LIN {X 0,Y 210.251,Z 700.702,A -85,B 0,C 180,E1 -22995.332,E2 -22995.332} C_VEL
LIN {X 0,Y 214.352,Z 687.95,A -85,B 0,C 180,E1 -22996.849,E2 -22996.849} C_VEL
LIN {X 0,Y 218.161,Z 673.656,A -85,B 0,C 180,E1 -22998.16,E2 -22998.16} C_VEL
LIN {X 0,Y 221.431,Z 658.156,A -85,B 0,C 180,E1 -22999.184,E2 -22999.184} C_VEL
LIN {X 0,Y 223.658,Z 642.562,A -85,B 0,C 180,E1 -22999.906,E2 -22999.906} C_VEL
LIN {X 0,Y 226.97,Z 599.755,A -85,B 0,C 180,E1 -23001.093,E2 -23001.093} C_VEL
LIN {X 0,Y 231.508,Z 536.215,A -85,B 0,C 180,E1 -23002.81,E2 -23002.81} C_VEL
LIN {X 0,Y 227.705,Z 547.018,A -85,B 0,C 180,E1 -23003.519,E2 -23003.519} C_VEL
LIN {X 0,Y 224.351,Z 554.465,A -85,B 0,C 180,E1 -23004.286,E2 -23004.286} C_VEL
LIN {X 0,Y 221.827,Z 558.997,A -85,B 0,C 180,E1 -23004.947,E2 -23004.947} C_VEL
LIN {X 0,Y 218.482,Z 569.62,A -85,B 0,C 180,E1 -23005.602,E2 -23005.602} C_VEL
LIN {X 0,Y 214.3,Z 580.329,A -85,B 0,C 180,E1 -23006.618,E2 -23006.618} C_VEL
LIN {X 0,Y 211.018,Z 586.681,A -85,B 0,C 180,E1 -23007.591,E2 -23007.591} C_VEL
LIN {X 0,Y 207.371,Z 592.159,A -85,B 0,C 180,E1 -23008.845,E2 -23008.845} C_VEL
LIN {X 0,Y 202.486,Z 604.004,A -85,B 0,C 180,E1 -23010.358,E2 -23010.358} C_VEL
LIN {X 0,Y 198.444,Z 611.857,A -85,B 0,C 180,E1 -23011.87,E2 -23011.87} C_VEL
LIN {X 0,Y 195.689,Z 615.882,A -85,B 0,C 180,E1 -23013.088,E2 -23013.088} C_VEL
LIN {X 0,Y 193.642,Z 618.166,A -85,B 0,C 180,E1 -23014.109,E2 -23014.109} C_VEL
LIN {X 0,Y 188.326,Z 629.557,A -85,B 0,C 180,E1 -23016.557,E2 -23016.557} C_VEL
LIN {X 0,Y 184.596,Z 636.026,A -85,B 0,C 180,E1 -23018.65,E2 -23018.65} C_VEL
LIN {X 0,Y 182.318,Z 638.821,A -85,B 0,C 180,E1 -23020.141,E2 -23020.141} C_VEL
LIN {X 0,Y 181.292,Z 639.784,A -85,B 0,C 180,E1 -23020.907,E2 -23020.907} C_VEL
LIN {X 0,Y 176.313,Z 648.748,A -85,B 0,C 180,E1 -23024.169,E2 -23024.169} C_VEL
LIN {X 0,Y 174.21,Z 651.8,A -85,B 0,C 180,E1 -23025.843,E2 -23025.843} C_VEL
LIN {X 0,Y 172.64,Z 653.404,A -85,B 0,C 180,E1 -23027.574,E2 -23027.574} C_VEL
LIN {X 0,Y 172.227,Z 654.518,A -85,B 0,C 180,E1 -23028.565,E2 -23028.565} C_VEL
LIN {X 0,Y 171.953,Z 657.794,A -85,B 0,C 180,E1 -23030.105,E2 -23030.105} C_VEL
LIN {X 0,Y 171.337,Z 668.465,A -85,B 0,C 180,E1 -23034.704,E2 -23034.704} C_VEL
LIN {X 0,Y 171.507,Z 677.415,A -85,B 0,C 180,E1 -23039.413,E2 -23039.413} C_VEL
LIN {X 0,Y 172.531,Z 684.128,A -85,B 0,C 180,E1 -23043.703,E2 -23043.703} C_VEL
LIN {X 0,Y 174.42,Z 689.78,A -85,B 0,C 180,E1 -23048.107,E2 -23048.107} C_VEL
LIN {X 0,Y 177.431,Z 694.715,A -85,B 0,C 180,E1 -23052.999,E2 -23052.999} C_VEL
LIN {X 0,Y 178.253,Z 696.265,A -85,B 0,C 180,E1 -23054.816,E2 -23054.816} C_VEL
LIN {X 0,Y 178.345,Z 698.551,A -85,B 0,C 180,E1 -23057.915,E2 -23057.915} C_VEL
LIN {X 0,Y 178.738,Z 700.109,A -85,B 0,C 180,E1 -23060.407,E2 -23060.407} C_VEL
LIN {X 0,Y 180.047,Z 701.114,A -85,B 0,C 180,E1 -23062.217,E2 -23062.217} C_VEL
LIN {X 0,Y 180.776,Z 701.337,A -85,B 0,C 180,E1 -23062.789,E2 -23062.789} C_VEL
LIN {X 0,Y 187.3,Z 702.48,A -85,B 0,C 180,E1 -23066.761,E2 -23066.761} C_VEL
LIN {X 0,Y 194.619,Z 702.496,A -85,B 0,C 180,E1 -23070.368,E2 -23070.368} C_VEL
LIN {X 0,Y 202.829,Z 701.412,A -85,B 0,C 180,E1 -23073.669,E2 -23073.669} C_VEL
LIN {X 0,Y 211.766,Z 699.284,A -85,B 0,C 180,E1 -23076.682,E2 -23076.682} C_VEL
LIN {X 0,Y 221.451,Z 696.077,A -85,B 0,C 180,E1 -23079.399,E2 -23079.399} C_VEL
LIN {X 0,Y 220.156,Z 697.084,A -85,B 0,C 180,E1 -23079.987,E2 -23079.987} C_VEL
LIN {X 0,Y 209.505,Z 703.658,A -85,B 0,C 180,E1 -23082.435,E2 -23082.435} C_VEL
LIN {X 0,Y 202.185,Z 708.181,A -85,B 0,C 180,E1 -23084.551,E2 -23084.551} C_VEL
LIN {X 0,Y 196.039,Z 722.236,A -85,B 0,C 180,E1 -23087.063,E2 -23087.063} C_VEL
LIN {X 0,Y 190.387,Z 733.904,A -85,B 0,C 180,E1 -23089.756,E2 -23089.756} C_VEL
LIN {X 0,Y 185.104,Z 743.709,A -85,B 0,C 180,E1 -23092.588,E2 -23092.588} C_VEL
LIN {X 0,Y 179.76,Z 753.29,A -85,B 0,C 180,E1 -23096.139,E2 -23096.139} C_VEL
LIN {X 0,Y 174.895,Z 761.263,A -85,B 0,C 180,E1 -23099.844,E2 -23099.844} C_VEL
LIN {X 0,Y 170.298,Z 768.682,A -85,B 0,C 180,E1 -23104.318,E2 -23104.318} C_VEL
LIN {X 0,Y 166.744,Z 774.56,A -85,B 0,C 180,E1 -23109.003,E2 -23109.003} C_VEL
LIN {X 0,Y 164.77,Z 778.036,A -85,B 0,C 180,E1 -23112.624,E2 -23112.624} C_VEL
LIN {X 0,Y 162.943,Z 781.562,A -85,B 0,C 180,E1 -23117.542,E2 -23117.542} C_VEL
LIN {X 0,Y 162.019,Z 783.877,A -85,B 0,C 180,E1 -23122.519,E2 -23122.519} C_VEL
LIN {X 0,Y 161.796,Z 785.034,A -85,B 0,C 180,E1 -23127.507,E2 -23127.507} C_VEL
LIN {X 0,Y 161.847,Z 785.184,A -85,B 0,C 180,E1 -23129.996,E2 -23129.996} C_VEL
LIN {X 0,Y 161.848,Z 784.583,A -85,B 0,C 180,E1 -23134.978,E2 -23134.978} C_VEL
LIN {X 0,Y 162.374,Z 782.833,A -85,B 0,C 180,E1 -23139.966,E2 -23139.966} C_VEL
LIN {X 0,Y 163.668,Z 779.907,A -85,B 0,C 180,E1 -23144.926,E2 -23144.926} C_VEL
LIN {X 0,Y 165.995,Z 775.732,A -85,B 0,C 180,E1 -23149.794,E2 -23149.794} C_VEL
LIN {X 0,Y 169.284,Z 770.198,A -85,B 0,C 180,E1 -23154.525,E2 -23154.525} C_VEL
LIN {X 0,Y 173.59,Z 763.151,A -85,B 0,C 180,E1 -23159.063,E2 -23159.063} C_VEL
LIN {X 0,Y 178.266,Z 755.599,A -85,B 0,C 180,E1 -23162.821,E2 -23162.821} C_VEL
LIN {X 0,Y 182.965,Z 747.147,A -85,B 0,C 180,E1 -23166.231,E2 -23166.231} C_VEL
LIN {X 0,Y 188.506,Z 737.217,A -85,B 0,C 180,E1 -23169.326,E2 -23169.326} C_VEL
LIN {X 0,Y 194.549,Z 725.183,A -85,B 0,C 180,E1 -23172.28,E2 -23172.28} C_VEL
LIN {X 0,Y 200.03,Z 712.892,A -85,B 0,C 180,E1 -23174.638,E2 -23174.638} C_VEL
LIN {X 0,Y 204.98,Z 700.094,A -85,B 0,C 180,E1 -23176.577,E2 -23176.577} C_VEL
LIN {X 0,Y 209.55,Z 685.921,A -85,B 0,C 180,E1 -23178.26,E2 -23178.26} C_VEL
LIN {X 0,Y 213.506,Z 671.096,A -85,B 0,C 180,E1 -23179.565,E2 -23179.565} C_VEL
LIN {X 0,Y 216.574,Z 656.308,A -85,B 0,C 180,E1 -23180.503,E2 -23180.503} C_VEL
LIN {X 0,Y 218.718,Z 641.008,A -85,B 0,C 180,E1 -23181.184,E2 -23181.184} C_VEL
LIN {X 0,Y 225.151,Z 556.647,A -85,B 0,C 180,E1 -23183.486,E2 -23183.486} C_VEL
LIN {X 0,Y 227.214,Z 528.253,A -85,B 0,C 180,E1 -23184.267,E2 -23184.267} C_VEL
LIN {X 0,Y 226.392,Z 506.219,A -85,B 0,C 180,E1 -23185.76,E2 -23185.76} C_VEL
LIN {X 0,Y 222.6,Z 494.178,A -85,B 0,C 180,E1 -23187.939,E2 -23187.939} C_VEL
LIN {X 0,Y 216.782,Z 485.116,A -85,B 0,C 180,E1 -23191.102,E2 -23191.102} C_VEL
LIN {X 0,Y 211.639,Z 478.028,A -85,B 0,C 180,E1 -23194.288,E2 -23194.288} C_VEL
LIN {X 0,Y 206.842,Z 471.641,A -85,B 0,C 180,E1 -23197.79,E2 -23197.79} C_VEL
LIN {X 0,Y 204.03,Z 467.883,A -85,B 0,C 180,E1 -23200.376,E2 -23200.376} C_VEL
LIN {X 0,Y 200.72,Z 462.777,A -85,B 0,C 180,E1 -23205.813,E2 -23205.813} C_VEL
LIN {X 0,Y 199.289,Z 459.944,A -85,B 0,C 180,E1 -23209.844,E2 -23209.844} C_VEL
LIN {X 0,Y 198.506,Z 458.911,A -85,B 0,C 180,E1 -23212.417,E2 -23212.417} C_VEL
LIN {X 0,Y 197.556,Z 457.928,A -85,B 0,C 180,E1 -23217.961,E2 -23217.961} C_VEL
LIN {X 0,Y 197.56,Z 458.311,A -85,B 0,C 180,E1 -23222.039,E2 -23222.039} C_VEL
LIN {X 0,Y 197.914,Z 459.91,A -85,B 0,C 180,E1 -23226.162,E2 -23226.162} C_VEL
LIN {X 0,Y 198.663,Z 462.572,A -85,B 0,C 180,E1 -23230.188,E2 -23230.188} C_VEL
LIN {X 0,Y 200.379,Z 467.163,A -85,B 0,C 180,E1 -23235.268,E2 -23235.268} C_VEL
LIN {X 0,Y 201.179,Z 469.388,A -85,B 0,C 180,E1 -23237.274,E2 -23237.274} C_VEL
LIN {X 0,Y 205.838,Z 476.9,A -85,B 0,C 180,E1 -23241.771,E2 -23241.771} C_VEL
LIN {X 0,Y 210.16,Z 484.065,A -85,B 0,C 180,E1 -23245.108,E2 -23245.108} C_VEL
LIN {X 0,Y 214.103,Z 491.145,A -85,B 0,C 180,E1 -23247.765,E2 -23247.765} C_VEL
LIN {X 0,Y 219.176,Z 501.028,A -85,B 0,C 180,E1 -23250.801,E2 -23250.801} C_VEL
LIN {X 0,Y 224.039,Z 511.702,A -85,B 0,C 180,E1 -23253.431,E2 -23253.431} C_VEL
LIN {X 0,Y 226.142,Z 516.859,A -85,B 0,C 180,E1 -23254.51,E2 -23254.51} C_VEL
LIN {X 0,Y 227.176,Z 535.771,A -85,B 0,C 180,E1 -23255.895,E2 -23255.895} C_VEL
LIN {X 0,Y 219.931,Z 632.241,A -85,B 0,C 180,E1 -23258.478,E2 -23258.478} C_VEL
LIN {X 0,Y 218.277,Z 648.104,A -85,B 0,C 180,E1 -23259.04,E2 -23259.04} C_VEL
LIN {X 0,Y 215.641,Z 663.359,A -85,B 0,C 180,E1 -23259.837,E2 -23259.837} C_VEL
LIN {X 0,Y 212.143,Z 678.063,A -85,B 0,C 180,E1 -23260.915,E2 -23260.915} C_VEL
LIN {X 0,Y 208.143,Z 691.846,A -85,B 0,C 180,E1 -23262.304,E2 -23262.304} C_VEL
LIN {X 0,Y 203.761,Z 704.529,A -85,B 0,C 180,E1 -23263.95,E2 -23263.95} C_VEL
LIN {X 0,Y 198.585,Z 717.228,A -85,B 0,C 180,E1 -23266.015,E2 -23266.015} C_VEL
LIN {X 0,Y 193.168,Z 728.856,A -85,B 0,C 180,E1 -23268.4,E2 -23268.4} C_VEL
LIN {X 0,Y 187.696,Z 739.514,A -85,B 0,C 180,E1 -23271.163,E2 -23271.163} C_VEL
LIN {X 0,Y 183.075,Z 747.963,A -85,B 0,C 180,E1 -23273.874,E2 -23273.874} C_VEL
LIN {X 0,Y 178.335,Z 756.228,A -85,B 0,C 180,E1 -23277.193,E2 -23277.193} C_VEL
LIN {X 0,Y 173.647,Z 763.764,A -85,B 0,C 180,E1 -23280.948,E2 -23280.948} C_VEL
LIN {X 0,Y 169.33,Z 770.801,A -85,B 0,C 180,E1 -23285.482,E2 -23285.482} C_VEL
LIN {X 0,Y 166.033,Z 776.334,A -85,B 0,C 180,E1 -23290.211,E2 -23290.211} C_VEL
LIN {X 0,Y 163.641,Z 780.512,A -85,B 0,C 180,E1 -23295.071,E2 -23295.071} C_VEL
LIN {X 0,Y 162.31,Z 783.445,A -85,B 0,C 180,E1 -23300.03,E2 -23300.03} C_VEL
LIN {X 0,Y 161.754,Z 785.206,A -85,B 0,C 180,E1 -23305.019,E2 -23305.019} C_VEL
LIN {X 0,Y 161.773,Z 785.815,A -85,B 0,C 180,E1 -23310.004,E2 -23310.004} C_VEL
LIN {X 0,Y 161.756,Z 785.237,A -85,B 0,C 180,E1 -23314.989,E2 -23314.989} C_VEL
LIN {X 0,Y 162.312,Z 783.519,A -85,B 0,C 180,E1 -23319.978,E2 -23319.978} C_VEL
LIN {X 0,Y 163.63,Z 780.622,A -85,B 0,C 180,E1 -23324.938,E2 -23324.938} C_VEL
LIN {X 0,Y 165.983,Z 776.481,A -85,B 0,C 180,E1 -23329.803,E2 -23329.803} C_VEL
LIN {X 0,Y 169.289,Z 770.996,A -85,B 0,C 180,E1 -23334.532,E2 -23334.532} C_VEL
LIN {X 0,Y 173.575,Z 764.013,A -85,B 0,C 180,E1 -23339.074,E2 -23339.074} C_VEL
LIN {X 0,Y 178.256,Z 756.526,A -85,B 0,C 180,E1 -23342.831,E2 -23342.831} C_VEL
LIN {X 0,Y 183.478,Z 747.452,A -85,B 0,C 180,E1 -23346.448,E2 -23346.448} C_VEL
LIN {X 0,Y 188.503,Z 738.293,A -85,B 0,C 180,E1 -23349.336,E2 -23349.336} C_VEL
LIN {X 0,Y 194.503,Z 726.418,A -85,B 0,C 180,E1 -23352.301,E2 -23352.301} C_VEL
LIN {X 0,Y 200.016,Z 714.299,A -85,B 0,C 180,E1 -23354.651,E2 -23354.651} C_VEL
LIN {X 0,Y 204.979,Z 701.582,A -85,B 0,C 180,E1 -23356.621,E2 -23356.621} C_VEL
LIN {X 0,Y 209.551,Z 687.912,A -85,B 0,C 180,E1 -23358.268,E2 -23358.268} C_VEL
LIN {X 0,Y 213.203,Z 674.707,A -85,B 0,C 180,E1 -23359.488,E2 -23359.488} C_VEL
LIN {X 0,Y 216.425,Z 660.328,A -85,B 0,C 180,E1 -23360.469,E2 -23360.469} C_VEL
LIN {X 0,Y 218.708,Z 645.822,A -85,B 0,C 180,E1 -23361.196,E2 -23361.196} C_VEL
LIN {X 0,Y 220.419,Z 628.463,A -85,B 0,C 180,E1 -23361.739,E2 -23361.739} C_VEL
LIN {X 0,Y 225.334,Z 562.086,A -85,B 0,C 180,E1 -23363.54,E2 -23363.54} C_VEL
LIN {X 0,Y 221.634,Z 573.32,A -85,B 0,C 180,E1 -23364.234,E2 -23364.234} C_VEL
LIN {X 0,Y 217.304,Z 584.041,A -85,B 0,C 180,E1 -23365.23,E2 -23365.23} C_VEL
LIN {X 0,Y 213.868,Z 590.614,A -85,B 0,C 180,E1 -23366.182,E2 -23366.182} C_VEL
LIN {X 0,Y 210.421,Z 595.815,A -85,B 0,C 180,E1 -23367.279,E2 -23367.279} C_VEL
LIN {X 0,Y 209.547,Z 597.49,A -85,B 0,C 180,E1 -23367.546,E2 -23367.546} C_VEL
LIN {X 0,Y 204.791,Z 608.486,A -85,B 0,C 180,E1 -23368.951,E2 -23368.951} C_VEL
LIN {X 0,Y 200.331,Z 616.846,A -85,B 0,C 180,E1 -23370.526,E2 -23370.526} C_VEL
LIN {X 0,Y 197.026,Z 621.56,A -85,B 0,C 180,E1 -23371.905,E2 -23371.905} C_VEL
LIN {X 0,Y 194.971,Z 624.011,A -85,B 0,C 180,E1 -23372.857,E2 -23372.857} C_VEL
LIN {X 0,Y 189.487,Z 635.143,A -85,B 0,C 180,E1 -23375.256,E2 -23375.256} C_VEL
LIN {X 0,Y 185.24,Z 641.839,A -85,B 0,C 180,E1 -23377.409,E2 -23377.409} C_VEL
LIN {X 0,Y 182.479,Z 645.036,A -85,B 0,C 180,E1 -23379.046,E2 -23379.046} C_VEL
LIN {X 0,Y 181.132,Z 646.367,A -85,B 0,C 180,E1 -23379.931,E2 -23379.931} C_VEL
LIN {X 0,Y 176.914,Z 653.338,A -85,B 0,C 180,E1 -23382.325,E2 -23382.325} C_VEL
LIN {X 0,Y 173.915,Z 657.504,A -85,B 0,C 180,E1 -23384.396,E2 -23384.396} C_VEL
LIN {X 0,Y 171.706,Z 659.762,A -85,B 0,C 180,E1 -23386.351,E2 -23386.351} C_VEL
LIN {X 0,Y 170.642,Z 660.646,A -85,B 0,C 180,E1 -23387.494,E2 -23387.494} C_VEL
LIN {X 0,Y 166.279,Z 667.419,A -85,B 0,C 180,E1 -23391.493,E2 -23391.493} C_VEL
LIN {X 0,Y 165.327,Z 668.75,A -85,B 0,C 180,E1 -23392.673,E2 -23392.673} C_VEL
LIN {X 0,Y 164.402,Z 669.807,A -85,B 0,C 180,E1 -23394.48,E2 -23394.48} C_VEL
LIN {X 0,Y 164.259,Z 670.417,A -85,B 0,C 180,E1 -23395.552,E2 -23395.552} C_VEL
LIN {X 0,Y 164.286,Z 673.502,A -85,B 0,C 180,E1 -23397.548,E2 -23397.548} C_VEL
LIN {X 0,Y 164.95,Z 681.681,A -85,B 0,C 180,E1 -23402.442,E2 -23402.442} C_VEL
LIN {X 0,Y 166.832,Z 688.336,A -85,B 0,C 180,E1 -23407.26,E2 -23407.26} C_VEL
LIN {X 0,Y 169.411,Z 693.597,A -85,B 0,C 180,E1 -23411.971,E2 -23411.971} C_VEL
LIN {X 0,Y 173.203,Z 697.589,A -85,B 0,C 180,E1 -23416.501,E2 -23416.501} C_VEL
LIN {X 0,Y 178.048,Z 700.399,A -85,B 0,C 180,E1 -23420.809,E2 -23420.809} C_VEL
LIN {X 0,Y 180.776,Z 701.337,A -85,B 0,C 180,E1 -23422.789,E2 -23422.789} C_VEL
LIN {X 0,Y 182.713,Z 702.165,A -85,B 0,C 180,E1 -23424.531,E2 -23424.531} C_VEL
LIN {X 0,Y 185.561,Z 703.804,A -85,B 0,C 180,E1 -23428.727,E2 -23428.727} C_VEL
LIN {X 0,Y 188.138,Z 704.229,A -85,B 0,C 180,E1 -23431.004,E2 -23431.004} C_VEL
LIN {X 0,Y 190.144,Z 704.213,A -85,B 0,C 180,E1 -23432.024,E2 -23432.024} C_VEL
LIN {X 0,Y 197.24,Z 703.639,A -85,B 0,C 180,E1 -23434.757,E2 -23434.757} C_VEL
LIN {X 0,Y 206.502,Z 701.978,A -85,B 0,C 180,E1 -23437.778,E2 -23437.778} C_VEL
LIN {X 0,Y 211.407,Z 700.744,A -85,B 0,C 180,E1 -23439.171,E2 -23439.171} C_VEL
LIN {X 0,Y 210.172,Z 701.567,A -85,B 0,C 180,E1 -23439.723,E2 -23439.723} C_VEL
LIN {X 0,Y 199.698,Z 707.167,A -85,B 0,C 180,E1 -23442.345,E2 -23442.345} C_VEL
LIN {X 0,Y 196.991,Z 708.851,A -85,B 0,C 180,E1 -23443.181,E2 -23443.181} C_VEL
LIN {X 0,Y 190.885,Z 722.261,A -85,B 0,C 180,E1 -23445.606,E2 -23445.606} C_VEL
LIN {X 0,Y 185.012,Z 733.926,A -85,B 0,C 180,E1 -23448.332,E2 -23448.332} C_VEL
LIN {X 0,Y 179.485,Z 743.73,A -85,B 0,C 180,E1 -23451.204,E2 -23451.204} C_VEL
LIN {X 0,Y 173.867,Z 753.309,A -85,B 0,C 180,E1 -23454.826,E2 -23454.826} C_VEL
LIN {X 0,Y 168.741,Z 761.281,A -85,B 0,C 180,E1 -23458.622,E2 -23458.622} C_VEL
LIN {X 0,Y 163.886,Z 768.699,A -85,B 0,C 180,E1 -23463.235,E2 -23463.235} C_VEL
LIN {X 0,Y 160.084,Z 774.576,A -85,B 0,C 180,E1 -23468.085,E2 -23468.085} C_VEL
LIN {X 0,Y 157.945,Z 778.051,A -85,B 0,C 180,E1 -23471.848,E2 -23471.848} C_VEL
LIN {X 0,Y 155.964,Z 781.577,A -85,B 0,C 180,E1 -23476.975,E2 -23476.975} C_VEL
LIN {X 0,Y 154.962,Z 783.891,A -85,B 0,C 180,E1 -23482.176,E2 -23482.176} C_VEL
LIN {X 0,Y 154.698,Z 785.048,A -85,B 0,C 180,E1 -23487.392,E2 -23487.392} C_VEL
LIN {X 0,Y 154.745,Z 785.198,A -85,B 0,C 180,E1 -23489.996,E2 -23489.996} C_VEL
LIN {X 0,Y 154.752,Z 784.597,A -85,B 0,C 180,E1 -23495.207,E2 -23495.207} C_VEL
LIN {X 0,Y 155.368,Z 782.847,A -85,B 0,C 180,E1 -23500.42,E2 -23500.42} C_VEL
LIN {X 0,Y 156.768,Z 779.92,A -85,B 0,C 180,E1 -23505.599,E2 -23505.599} C_VEL
LIN {X 0,Y 159.268,Z 775.746,A -85,B 0,C 180,E1 -23510.667,E2 -23510.667} C_VEL
LIN {X 0,Y 162.789,Z 770.212,A -85,B 0,C 180,E1 -23515.572,E2 -23515.572} C_VEL
LIN {X 0,Y 167.379,Z 763.166,A -85,B 0,C 180,E1 -23520.251,E2 -23520.251} C_VEL
LIN {X 0,Y 172.314,Z 755.614,A -85,B 0,C 180,E1 -23524.107,E2 -23524.107} C_VEL
LIN {X 0,Y 177.651,Z 746.518,A -85,B 0,C 180,E1 -23527.813,E2 -23527.813} C_VEL
LIN {X 0,Y 183.053,Z 737.234,A -85,B 0,C 180,E1 -23530.739,E2 -23530.739} C_VEL
LIN {X 0,Y 189.336,Z 725.202,A -85,B 0,C 180,E1 -23533.731,E2 -23533.731} C_VEL
LIN {X 0,Y 195.03,Z 712.913,A -85,B 0,C 180,E1 -23536.108,E2 -23536.108} C_VEL
LIN {X 0,Y 200.41,Z 699.424,A -85,B 0,C 180,E1 -23538.143,E2 -23538.143} C_VEL
LIN {X 0,Y 204.891,Z 685.95,A -85,B 0,C 180,E1 -23539.741,E2 -23539.741} C_VEL
LIN {X 0,Y 208.972,Z 671.133,A -85,B 0,C 180,E1 -23541.047,E2 -23541.047} C_VEL
LIN {X 0,Y 212.142,Z 656.359,A -85,B 0,C 180,E1 -23541.979,E2 -23541.979} C_VEL
LIN {X 0,Y 214.346,Z 641.09,A -85,B 0,C 180,E1 -23542.66,E2 -23542.66} C_VEL
LIN {X 0,Y 220.651,Z 561.424,A -85,B 0,C 180,E1 -23544.836,E2 -23544.836} C_VEL
LIN {X 0,Y 223.085,Z 528.82,A -85,B 0,C 180,E1 -23545.744,E2 -23545.744} C_VEL
LIN {X 0,Y 222.419,Z 509.121,A -85,B 0,C 180,E1 -23547.131,E2 -23547.131} C_VEL
LIN {X 0,Y 219.435,Z 499.25,A -85,B 0,C 180,E1 -23548.973,E2 -23548.973} C_VEL
LIN {X 0,Y 214.194,Z 490.861,A -85,B 0,C 180,E1 -23551.983,E2 -23551.983} C_VEL
LIN {X 0,Y 209.616,Z 484.382,A -85,B 0,C 180,E1 -23554.958,E2 -23554.958} C_VEL
LIN {X 0,Y 204.971,Z 477.997,A -85,B 0,C 180,E1 -23558.51,E2 -23558.51} C_VEL
LIN {X 0,Y 201.233,Z 473.311,A -85,B 0,C 180,E1 -23561.944,E2 -23561.944} C_VEL
LIN {X 0,Y 197.097,Z 468.223,A -85,B 0,C 180,E1 -23567.123,E2 -23567.123} C_VEL
LIN {X 0,Y 196.161,Z 466.455,A -85,B 0,C 180,E1 -23569.681,E2 -23569.681} C_VEL
LIN {X 0,Y 195.501,Z 465.473,A -85,B 0,C 180,E1 -23571.733,E2 -23571.733} C_VEL
LIN {X 0,Y 194.339,Z 464.264,A -85,B 0,C 180,E1 -23577.928,E2 -23577.928} C_VEL
LIN {X 0,Y 194.278,Z 464.276,A -85,B 0,C 180,E1 -23580,E2 -23580} C_VEL
LIN {X 0,Y 194.405,Z 465.29,A -85,B 0,C 180,E1 -23584.146,E2 -23584.146} C_VEL
LIN {X 0,Y 194.891,Z 467.577,A -85,B 0,C 180,E1 -23588.294,E2 -23588.294} C_VEL
LIN {X 0,Y 195.786,Z 469.986,A -85,B 0,C 180,E1 -23591.387,E2 -23591.387} C_VEL
LIN {X 0,Y 199.688,Z 476.11,A -85,B 0,C 180,E1 -23596.748,E2 -23596.748} C_VEL
LIN {X 0,Y 203.897,Z 483.123,A -85,B 0,C 180,E1 -23600.976,E2 -23600.976} C_VEL
LIN {X 0,Y 207.93,Z 490.091,A -85,B 0,C 180,E1 -23604.269,E2 -23604.269} C_VEL
LIN {X 0,Y 212.054,Z 497.752,A -85,B 0,C 180,E1 -23607.182,E2 -23607.182} C_VEL
LIN {X 0,Y 216.894,Z 507.782,A -85,B 0,C 180,E1 -23610.216,E2 -23610.216} C_VEL
LIN {X 0,Y 221.471,Z 518.344,A -85,B 0,C 180,E1 -23612.806,E2 -23612.806} C_VEL
LIN {X 0,Y 222.265,Z 520.724,A -85,B 0,C 180,E1 -23613.258,E2 -23613.258} C_VEL
LIN {X 0,Y 223.017,Z 536.645,A -85,B 0,C 180,E1 -23614.447,E2 -23614.447} C_VEL
LIN {X 0,Y 215.309,Z 635.545,A -85,B 0,C 180,E1 -23617.097,E2 -23617.097} C_VEL
LIN {X 0,Y 213.427,Z 651.168,A -85,B 0,C 180,E1 -23617.696,E2 -23617.696} C_VEL
LIN {X 0,Y 210.603,Z 666.177,A -85,B 0,C 180,E1 -23618.55,E2 -23618.55} C_VEL
LIN {X 0,Y 206.71,Z 681.204,A -85,B 0,C 180,E1 -23619.72,E2 -23619.72} C_VEL
LIN {X 0,Y 202.461,Z 694.771,A -85,B 0,C 180,E1 -23621.166,E2 -23621.166} C_VEL
LIN {X 0,Y 197.829,Z 707.309,A -85,B 0,C 180,E1 -23622.891,E2 -23622.891} C_VEL
LIN {X 0,Y 191.95,Z 720.646,A -85,B 0,C 180,E1 -23625.191,E2 -23625.191} C_VEL
LIN {X 0,Y 185.959,Z 732.637,A -85,B 0,C 180,E1 -23627.874,E2 -23627.874} C_VEL
LIN {X 0,Y 180.413,Z 742.711,A -85,B 0,C 180,E1 -23630.732,E2 -23630.732} C_VEL
LIN {X 0,Y 175.485,Z 751.216,A -85,B 0,C 180,E1 -23633.797,E2 -23633.797} C_VEL
LIN {X 0,Y 170.079,Z 759.604,A -85,B 0,C 180,E1 -23637.513,E2 -23637.513} C_VEL
LIN {X 0,Y 165.012,Z 767.468,A -85,B 0,C 180,E1 -23642.068,E2 -23642.068} C_VEL
LIN {X 0,Y 160.986,Z 773.732,A -85,B 0,C 180,E1 -23646.869,E2 -23646.869} C_VEL
LIN {X 0,Y 157.949,Z 778.571,A -85,B 0,C 180,E1 -23651.857,E2 -23651.857} C_VEL
LIN {X 0,Y 155.9,Z 782.115,A -85,B 0,C 180,E1 -23656.978,E2 -23656.978} C_VEL
LIN {X 0,Y 154.868,Z 784.456,A -85,B 0,C 180,E1 -23662.18,E2 -23662.18} C_VEL
LIN {X 0,Y 154.628,Z 785.644,A -85,B 0,C 180,E1 -23667.399,E2 -23667.399} C_VEL
LIN {X 0,Y 154.628,Z 785.772,A -85,B 0,C 180,E1 -23670.678,E2 -23670.678} C_VEL
LIN {X 0,Y 154.685,Z 785.223,A -85,B 0,C 180,E1 -23675.218,E2 -23675.218} C_VEL
LIN {X 0,Y 155.283,Z 783.505,A -85,B 0,C 180,E1 -23680.434,E2 -23680.434} C_VEL
LIN {X 0,Y 156.729,Z 780.607,A -85,B 0,C 180,E1 -23685.612,E2 -23685.612} C_VEL
LIN {X 0,Y 159.261,Z 776.465,A -85,B 0,C 180,E1 -23690.677,E2 -23690.677} C_VEL
LIN {X 0,Y 162.794,Z 770.979,A -85,B 0,C 180,E1 -23695.58,E2 -23695.58} C_VEL
LIN {X 0,Y 167.351,Z 763.995,A -85,B 0,C 180,E1 -23700.265,E2 -23700.265} C_VEL
LIN {X 0,Y 172.295,Z 756.507,A -85,B 0,C 180,E1 -23704.12,E2 -23704.12} C_VEL
LIN {X 0,Y 177.409,Z 748.048,A -85,B 0,C 180,E1 -23707.599,E2 -23707.599} C_VEL
LIN {X 0,Y 183.035,Z 738.27,A -85,B 0,C 180,E1 -23710.753,E2 -23710.753} C_VEL
LIN {X 0,Y 189.297,Z 726.393,A -85,B 0,C 180,E1 -23713.752,E2 -23713.752} C_VEL
LIN {X 0,Y 195.021,Z 714.27,A -85,B 0,C 180,E1 -23716.12,E2 -23716.12} C_VEL
LIN {X 0,Y 200.26,Z 701.308,A -85,B 0,C 180,E1 -23718.133,E2 -23718.133} C_VEL
LIN {X 0,Y 204.884,Z 687.873,A -85,B 0,C 180,E1 -23719.753,E2 -23719.753} C_VEL
LIN {X 0,Y 208.67,Z 674.659,A -85,B 0,C 180,E1 -23720.967,E2 -23720.967} C_VEL
LIN {X 0,Y 211.985,Z 660.266,A -85,B 0,C 180,E1 -23721.946,E2 -23721.946} C_VEL
LIN {X 0,Y 214.384,Z 645.385,A -85,B 0,C 180,E1 -23722.687,E2 -23722.687} C_VEL
LIN {X 0,Y 216.148,Z 627.699,A -85,B 0,C 180,E1 -23723.232,E2 -23723.232} C_VEL
LIN {X 0,Y 218.861,Z 592.58,A -85,B 0,C 180,E1 -23724.18,E2 -23724.18} C_VEL
LIN {X 0,Y 217.92,Z 592.739,A -85,B 0,C 180,E1 -23724.513,E2 -23724.513} C_VEL
LIN {X 0,Y 213.861,Z 599.214,A -85,B 0,C 180,E1 -23725.681,E2 -23725.681} C_VEL
LIN {X 0,Y 212.383,Z 601.438,A -85,B 0,C 180,E1 -23726.134,E2 -23726.134} C_VEL
LIN {X 0,Y 207.382,Z 612.649,A -85,B 0,C 180,E1 -23727.525,E2 -23727.525} C_VEL
LIN {X 0,Y 202.655,Z 621.279,A -85,B 0,C 180,E1 -23729.09,E2 -23729.09} C_VEL
LIN {X 0,Y 198.859,Z 626.745,A -85,B 0,C 180,E1 -23730.563,E2 -23730.563} C_VEL
LIN {X 0,Y 196.638,Z 629.386,A -85,B 0,C 180,E1 -23731.525,E2 -23731.525} C_VEL
LIN {X 0,Y 190.966,Z 640.095,A -85,B 0,C 180,E1 -23733.792,E2 -23733.792} C_VEL
LIN {X 0,Y 186.125,Z 647.178,A -85,B 0,C 180,E1 -23735.977,E2 -23735.977} C_VEL
LIN {X 0,Y 182.698,Z 651.019,A -85,B 0,C 180,E1 -23737.823,E2 -23737.823} C_VEL
LIN {X 0,Y 181.151,Z 652.533,A -85,B 0,C 180,E1 -23738.716,E2 -23738.716} C_VEL
LIN {X 0,Y 176.241,Z 659.754,A -85,B 0,C 180,E1 -23741.245,E2 -23741.245} C_VEL
LIN {X 0,Y 172.904,Z 663.809,A -85,B 0,C 180,E1 -23743.358,E2 -23743.358} C_VEL
LIN {X 0,Y 170.15,Z 666.365,A -85,B 0,C 180,E1 -23745.651,E2 -23745.651} C_VEL
LIN {X 0,Y 168.936,Z 667.469,A -85,B 0,C 180,E1 -23746.773,E2 -23746.773} C_VEL
LIN {X 0,Y 164.804,Z 673.237,A -85,B 0,C 180,E1 -23750.178,E2 -23750.178} C_VEL
LIN {X 0,Y 163.335,Z 675.053,A -85,B 0,C 180,E1 -23751.77,E2 -23751.77} C_VEL
LIN {X 0,Y 161.534,Z 676.871,A -85,B 0,C 180,E1 -23755.008,E2 -23755.008} C_VEL
LIN {X 0,Y 159.152,Z 681.134,A -85,B 0,C 180,E1 -23758.735,E2 -23758.735} C_VEL
LIN {X 0,Y 158.605,Z 682.241,A -85,B 0,C 180,E1 -23760,E2 -23760} C_VEL
LIN {X 0,Y 158.192,Z 683.809,A -85,B 0,C 180,E1 -23763.183,E2 -23763.183} C_VEL
LIN {X 0,Y 158.486,Z 684.399,A -85,B 0,C 180,E1 -23764.451,E2 -23764.451} C_VEL
LIN {X 0,Y 161.743,Z 692.448,A -85,B 0,C 180,E1 -23771.276,E2 -23771.276} C_VEL
LIN {X 0,Y 165.314,Z 697.111,A -85,B 0,C 180,E1 -23776.041,E2 -23776.041} C_VEL
LIN {X 0,Y 168.785,Z 699.826,A -85,B 0,C 180,E1 -23779.457,E2 -23779.457} C_VEL
LIN {X 0,Y 174.444,Z 702.402,A -85,B 0,C 180,E1 -23783.758,E2 -23783.758} C_VEL
LIN {X 0,Y 181.127,Z 703.869,A -85,B 0,C 180,E1 -23787.75,E2 -23787.75} C_VEL
LIN {X 0,Y 188.72,Z 704.28,A -85,B 0,C 180,E1 -23791.424,E2 -23791.424} C_VEL
LIN {X 0,Y 190.144,Z 704.213,A -85,B 0,C 180,E1 -23792.024,E2 -23792.024} C_VEL
LIN {X 0,Y 191.974,Z 704.312,A -85,B 0,C 180,E1 -23793.089,E2 -23793.089} C_VEL
LIN {X 0,Y 195.572,Z 705.196,A -85,B 0,C 180,E1 -23796.926,E2 -23796.926} C_VEL
LIN {X 0,Y 197.74,Z 705.017,A -85,B 0,C 180,E1 -23797.893,E2 -23797.893} C_VEL
LIN {X 0,Y 201.258,Z 704.484,A -85,B 0,C 180,E1 -23798.944,E2 -23798.944} C_VEL
LIN {X 0,Y 200.255,Z 705.124,A -85,B 0,C 180,E1 -23799.454,E2 -23799.454} C_VEL
LIN {X 0,Y 192.048,Z 709.215,A -85,B 0,C 180,E1 -23801.685,E2 -23801.685} C_VEL
LIN {X 0,Y 185.339,Z 723.345,A -85,B 0,C 180,E1 -23804.293,E2 -23804.293} C_VEL
LIN {X 0,Y 179.755,Z 733.949,A -85,B 0,C 180,E1 -23806.822,E2 -23806.822} C_VEL
LIN {X 0,Y 173.978,Z 743.75,A -85,B 0,C 180,E1 -23809.73,E2 -23809.73} C_VEL
LIN {X 0,Y 168.873,Z 752.103,A -85,B 0,C 180,E1 -23812.879,E2 -23812.879} C_VEL
LIN {X 0,Y 163.355,Z 760.267,A -85,B 0,C 180,E1 -23816.729,E2 -23816.729} C_VEL
LIN {X 0,Y 158.734,Z 767.009,A -85,B 0,C 180,E1 -23820.85,E2 -23820.85} C_VEL
LIN {X 0,Y 154.336,Z 773.247,A -85,B 0,C 180,E1 -23825.802,E2 -23825.802} C_VEL
LIN {X 0,Y 151.162,Z 778.066,A -85,B 0,C 180,E1 -23831.003,E2 -23831.003} C_VEL
LIN {X 0,Y 149.011,Z 781.592,A -85,B 0,C 180,E1 -23836.356,E2 -23836.356} C_VEL
LIN {X 0,Y 147.906,Z 783.905,A -85,B 0,C 180,E1 -23841.8,E2 -23841.8} C_VEL
LIN {X 0,Y 147.61,Z 785.062,A -85,B 0,C 180,E1 -23847.267,E2 -23847.267} C_VEL
LIN {X 0,Y 147.621,Z 785.144,A -85,B 0,C 180,E1 -23851.223,E2 -23851.223} C_VEL
LIN {X 0,Y 147.684,Z 784.611,A -85,B 0,C 180,E1 -23855.457,E2 -23855.457} C_VEL
LIN {X 0,Y 148.347,Z 782.86,A -85,B 0,C 180,E1 -23860.919,E2 -23860.919} C_VEL
LIN {X 0,Y 149.89,Z 779.934,A -85,B 0,C 180,E1 -23866.335,E2 -23866.335} C_VEL
LIN {X 0,Y 152.591,Z 775.76,A -85,B 0,C 180,E1 -23871.616,E2 -23871.616} C_VEL
LIN {X 0,Y 156.354,Z 770.226,A -85,B 0,C 180,E1 -23876.706,E2 -23876.706} C_VEL
LIN {X 0,Y 161.253,Z 763.18,A -85,B 0,C 180,E1 -23881.529,E2 -23881.529} C_VEL
LIN {X 0,Y 166.453,Z 755.629,A -85,B 0,C 180,E1 -23885.484,E2 -23885.484} C_VEL
LIN {X 0,Y 172.078,Z 746.53,A -85,B 0,C 180,E1 -23889.269,E2 -23889.269} C_VEL
LIN {X 0,Y 177.705,Z 737.251,A -85,B 0,C 180,E1 -23892.242,E2 -23892.242} C_VEL
LIN {X 0,Y 184.26,Z 725.221,A -85,B 0,C 180,E1 -23895.261,E2 -23895.261} C_VEL
LIN {X 0,Y 190.163,Z 712.934,A -85,B 0,C 180,E1 -23897.654,E2 -23897.654} C_VEL
LIN {X 0,Y 195.297,Z 700.604,A -85,B 0,C 180,E1 -23899.546,E2 -23899.546} C_VEL
LIN {X 0,Y 199.781,Z 687.802,A -85,B 0,C 180,E1 -23901.101,E2 -23901.101} C_VEL
LIN {X 0,Y 203.976,Z 673.543,A -85,B 0,C 180,E1 -23902.41,E2 -23902.41} C_VEL
LIN {X 0,Y 207.521,Z 658.084,A -85,B 0,C 180,E1 -23903.437,E2 -23903.437} C_VEL
LIN {X 0,Y 209.973,Z 642.53,A -85,B 0,C 180,E1 -23904.151,E2 -23904.151} C_VEL
LIN {X 0,Y 213.689,Z 598.892,A -85,B 0,C 180,E1 -23905.357,E2 -23905.357} C_VEL
LIN {X 0,Y 219.112,Z 529.846,A -85,B 0,C 180,E1 -23907.247,E2 -23907.247} C_VEL
LIN {X 0,Y 218.638,Z 512.259,A -85,B 0,C 180,E1 -23908.51,E2 -23908.51} C_VEL
LIN {X 0,Y 216.39,Z 504.4,A -85,B 0,C 180,E1 -23910.009,E2 -23910.009} C_VEL
LIN {X 0,Y 211.723,Z 496.702,A -85,B 0,C 180,E1 -23912.844,E2 -23912.844} C_VEL
LIN {X 0,Y 206.713,Z 489.371,A -85,B 0,C 180,E1 -23916.321,E2 -23916.321} C_VEL
LIN {X 0,Y 201.97,Z 482.784,A -85,B 0,C 180,E1 -23920.3,E2 -23920.3} C_VEL
LIN {X 0,Y 198.773,Z 478.841,A -85,B 0,C 180,E1 -23923.57,E2 -23923.57} C_VEL
LIN {X 0,Y 194.972,Z 474.075,A -85,B 0,C 180,E1 -23928.829,E2 -23928.829} C_VEL
LIN {X 0,Y 193.342,Z 472.146,A -85,B 0,C 180,E1 -23932.166,E2 -23932.166} C_VEL
LIN {X 0,Y 191.855,Z 470.925,A -85,B 0,C 180,E1 -23937.901,E2 -23937.901} C_VEL
LIN {X 0,Y 191.787,Z 471.218,A -85,B 0,C 180,E1 -23941.575,E2 -23941.575} C_VEL
LIN {X 0,Y 192.442,Z 472.8,A -85,B 0,C 180,E1 -23945.526,E2 -23945.526} C_VEL
LIN {X 0,Y 194.412,Z 476.479,A -85,B 0,C 180,E1 -23950.545,E2 -23950.545} C_VEL
LIN {X 0,Y 198.125,Z 482.542,A -85,B 0,C 180,E1 -23956.031,E2 -23956.031} C_VEL
LIN {X 0,Y 202.043,Z 489.434,A -85,B 0,C 180,E1 -23960.21,E2 -23960.21} C_VEL
LIN {X 0,Y 205.769,Z 496.098,A -85,B 0,C 180,E1 -23963.426,E2 -23963.426} C_VEL
LIN {X 0,Y 209.698,Z 503.781,A -85,B 0,C 180,E1 -23966.365,E2 -23966.365} C_VEL
LIN {X 0,Y 213.824,Z 512.687,A -85,B 0,C 180,E1 -23969.112,E2 -23969.112} C_VEL
LIN {X 0,Y 218.238,Z 523.263,A -85,B 0,C 180,E1 -23971.773,E2 -23971.773} C_VEL
LIN {X 0,Y 218.478,Z 524.516,A -85,B 0,C 180,E1 -23971.95,E2 -23971.95} C_VEL
LIN {X 0,Y 218.979,Z 537.8,A -85,B 0,C 180,E1 -23972.95,E2 -23972.95} C_VEL
LIN {X 0,Y 210.966,Z 636.877,A -85,B 0,C 180,E1 -23975.611,E2 -23975.611} C_VEL
LIN {X 0,Y 209.011,Z 651.991,A -85,B 0,C 180,E1 -23976.202,E2 -23976.202} C_VEL
LIN {X 0,Y 205.928,Z 667.398,A -85,B 0,C 180,E1 -23977.09,E2 -23977.09} C_VEL
LIN {X 0,Y 202.236,Z 681.174,A -85,B 0,C 180,E1 -23978.169,E2 -23978.169} C_VEL
LIN {X 0,Y 197.734,Z 695.043,A -85,B 0,C 180,E1 -23979.65,E2 -23979.65} C_VEL
LIN {X 0,Y 193.055,Z 707.287,A -85,B 0,C 180,E1 -23981.343,E2 -23981.343} C_VEL
LIN {X 0,Y 186.969,Z 720.626,A -85,B 0,C 180,E1 -23983.654,E2 -23983.654} C_VEL
LIN {X 0,Y 180.718,Z 732.62,A -85,B 0,C 180,E1 -23986.353,E2 -23986.353} C_VEL
LIN {X 0,Y 174.924,Z 742.695,A -85,B 0,C 180,E1 -23989.246,E2 -23989.246} C_VEL
LIN {X 0,Y 169.736,Z 751.201,A -85,B 0,C 180,E1 -23992.363,E2 -23992.363} C_VEL
LIN {X 0,Y 164.098,Z 759.589,A -85,B 0,C 180,E1 -23996.173,E2 -23996.173} C_VEL
LIN {X 0,Y 158.733,Z 767.454,A -85,B 0,C 180,E1 -24000.859,E2 -24000.859} C_VEL
LIN {X 0,Y 154.429,Z 773.718,A -85,B 0,C 180,E1 -24005.826,E2 -24005.826} C_VEL
LIN {X 0,Y 151.168,Z 778.557,A -85,B 0,C 180,E1 -24011.012,E2 -24011.012} C_VEL
LIN {X 0,Y 148.954,Z 782.101,A -85,B 0,C 180,E1 -24016.359,E2 -24016.359} C_VEL
LIN {X 0,Y 147.808,Z 784.442,A -85,B 0,C 180,E1 -24021.803,E2 -24021.803} C_VEL
LIN {X 0,Y 147.526,Z 785.63,A -85,B 0,C 180,E1 -24027.274,E2 -24027.274} C_VEL
LIN {X 0,Y 147.589,Z 785.787,A -85,B 0,C 180,E1 -24030.004,E2 -24030.004} C_VEL
LIN {X 0,Y 147.612,Z 785.209,A -85,B 0,C 180,E1 -24035.468,E2 -24035.468} C_VEL
LIN {X 0,Y 148.276,Z 783.49,A -85,B 0,C 180,E1 -24040.933,E2 -24040.933} C_VEL
LIN {X 0,Y 149.851,Z 780.592,A -85,B 0,C 180,E1 -24046.348,E2 -24046.348} C_VEL
LIN {X 0,Y 152.587,Z 776.45,A -85,B 0,C 180,E1 -24051.626,E2 -24051.626} C_VEL
LIN {X 0,Y 156.358,Z 770.963,A -85,B 0,C 180,E1 -24056.714,E2 -24056.714} C_VEL
LIN {X 0,Y 161.217,Z 763.977,A -85,B 0,C 180,E1 -24061.546,E2 -24061.546} C_VEL
LIN {X 0,Y 166.42,Z 756.488,A -85,B 0,C 180,E1 -24065.502,E2 -24065.502} C_VEL
LIN {X 0,Y 172.271,Z 747.257,A -85,B 0,C 180,E1 -24069.332,E2 -24069.332} C_VEL
LIN {X 0,Y 178.674,Z 736.549,A -85,B 0,C 180,E1 -24072.732,E2 -24072.732} C_VEL
LIN {X 0,Y 184.72,Z 725.326,A -85,B 0,C 180,E1 -24075.514,E2 -24075.514} C_VEL
LIN {X 0,Y 190.712,Z 712.99,A -85,B 0,C 180,E1 -24077.875,E2 -24077.875} C_VEL
LIN {X 0,Y 195.727,Z 700.91,A -85,B 0,C 180,E1 -24079.734,E2 -24079.734} C_VEL
LIN {X 0,Y 200.36,Z 687.834,A -85,B 0,C 180,E1 -24081.307,E2 -24081.307} C_VEL
LIN {X 0,Y 204.276,Z 674.612,A -85,B 0,C 180,E1 -24082.513,E2 -24082.513} C_VEL
LIN {X 0,Y 207.692,Z 660.205,A -85,B 0,C 180,E1 -24083.485,E2 -24083.485} C_VEL
LIN {X 0,Y 210.232,Z 644.891,A -85,B 0,C 180,E1 -24084.237,E2 -24084.237} C_VEL
LIN {X 0,Y 212.056,Z 626.644,A -85,B 0,C 180,E1 -24084.79,E2 -24084.79} C_VEL
LIN {X 0,Y 213.248,Z 610.193,A -85,B 0,C 180,E1 -24085.282,E2 -24085.282} C_VEL
LIN {X 0,Y 208.515,Z 619.796,A -85,B 0,C 180,E1 -24086.602,E2 -24086.602} C_VEL
LIN {X 0,Y 203.688,Z 627.953,A -85,B 0,C 180,E1 -24088.172,E2 -24088.172} C_VEL
LIN {X 0,Y 199.696,Z 633.172,A -85,B 0,C 180,E1 -24089.689,E2 -24089.689} C_VEL
LIN {X 0,Y 198.163,Z 635.159,A -85,B 0,C 180,E1 -24090.303,E2 -24090.303} C_VEL
LIN {X 0,Y 192.355,Z 645.206,A -85,B 0,C 180,E1 -24092.383,E2 -24092.383} C_VEL
LIN {X 0,Y 187.03,Z 652.445,A -85,B 0,C 180,E1 -24094.532,E2 -24094.532} C_VEL
LIN {X 0,Y 183.042,Z 656.693,A -85,B 0,C 180,E1 -24096.431,E2 -24096.431} C_VEL
LIN {X 0,Y 181.186,Z 658.468,A -85,B 0,C 180,E1 -24097.422,E2 -24097.422} C_VEL
LIN {X 0,Y 176.467,Z 664.749,A -85,B 0,C 180,E1 -24099.605,E2 -24099.605} C_VEL
LIN {X 0,Y 173.624,Z 668.088,A -85,B 0,C 180,E1 -24101.105,E2 -24101.105} C_VEL
LIN {X 0,Y 170.419,Z 671.227,A -85,B 0,C 180,E1 -24103.221,E2 -24103.221} C_VEL
LIN {X 0,Y 167.744,Z 673.403,A -85,B 0,C 180,E1 -24105.44,E2 -24105.44} C_VEL
LIN {X 0,Y 163.218,Z 678.967,A -85,B 0,C 180,E1 -24108.827,E2 -24108.827} C_VEL
LIN {X 0,Y 161.993,Z 680.344,A -85,B 0,C 180,E1 -24110.006,E2 -24110.006} C_VEL
LIN {X 0,Y 158.454,Z 684.045,A -85,B 0,C 180,E1 -24114.91,E2 -24114.91} C_VEL
LIN {X 0,Y 156.023,Z 687.964,A -85,B 0,C 180,E1 -24118.709,E2 -24118.709} C_VEL
LIN {X 0,Y 155.051,Z 690.086,A -85,B 0,C 180,E1 -24122.598,E2 -24122.598} C_VEL
LIN {X 0,Y 155.033,Z 690.605,A -85,B 0,C 180,E1 -24124.156,E2 -24124.156} C_VEL
LIN {X 0,Y 154.646,Z 693.329,A -85,B 0,C 180,E1 -24127.836,E2 -24127.836} C_VEL
LIN {X 0,Y 154.964,Z 694.806,A -85,B 0,C 180,E1 -24130.452,E2 -24130.452} C_VEL
LIN {X 0,Y 156.968,Z 696.294,A -85,B 0,C 180,E1 -24134.918,E2 -24134.918} C_VEL
LIN {X 0,Y 159.68,Z 698.44,A -85,B 0,C 180,E1 -24137.944,E2 -24137.944} C_VEL
LIN {X 0,Y 164.947,Z 701.955,A -85,B 0,C 180,E1 -24142.549,E2 -24142.549} C_VEL
LIN {X 0,Y 171.396,Z 704.396,A -85,B 0,C 180,E1 -24146.811,E2 -24146.811} C_VEL
LIN {X 0,Y 178.764,Z 705.722,A -85,B 0,C 180,E1 -24150.736,E2 -24150.736} C_VEL
LIN {X 0,Y 187.178,Z 705.972,A -85,B 0,C 180,E1 -24154.278,E2 -24154.278} C_VEL
LIN {X 0,Y 197.74,Z 705.017,A -85,B 0,C 180,E1 -24157.893,E2 -24157.893} C_VEL
LIN {X 0,Y 198.123,Z 705.177,A -85,B 0,C 180,E1 -24158.27,E2 -24158.27} C_VEL
LIN {X 0,Y 197.228,Z 706.094,A -85,B 0,C 180,E1 -24158.911,E2 -24158.911} C_VEL
LIN {X 0,Y 194.688,Z 707.771,A -85,B 0,C 180,E1 -24159.583,E2 -24159.583} C_VEL
LIN {X 0,Y 188.144,Z 711.898,A -85,B 0,C 180,E1 -24160.487,E2 -24160.487} C_VEL
LIN {X 0,Y 184.711,Z 715.204,A -85,B 0,C 180,E1 -24161.086,E2 -24161.086} C_VEL
LIN {X 0,Y 183.904,Z 716.513,A -85,B 0,C 180,E1 -24161.319,E2 -24161.319} C_VEL
LIN {X 0,Y 177.764,Z 728.408,A -85,B 0,C 180,E1 -24163.815,E2 -24163.815} C_VEL
LIN {X 0,Y 171.527,Z 739.074,A -85,B 0,C 180,E1 -24166.658,E2 -24166.658} C_VEL
LIN {X 0,Y 164.907,Z 749.452,A -85,B 0,C 180,E1 -24170.258,E2 -24170.258} C_VEL
LIN {X 0,Y 159.059,Z 758.069,A -85,B 0,C 180,E1 -24174.161,E2 -24174.161} C_VEL
LIN {X 0,Y 153.829,Z 765.23,A -85,B 0,C 180,E1 -24178.3,E2 -24178.3} C_VEL
LIN {X 0,Y 148.91,Z 771.852,A -85,B 0,C 180,E1 -24183.358,E2 -24183.358} C_VEL
LIN {X 0,Y 145.17,Z 777.023,A -85,B 0,C 180,E1 -24188.706,E2 -24188.706} C_VEL
LIN {X 0,Y 143.058,Z 780,A -85,B 0,C 180,E1 -24192.852,E2 -24192.852} C_VEL
LIN {X 0,Y 141.361,Z 782.911,A -85,B 0,C 180,E1 -24198.525,E2 -24198.525} C_VEL
LIN {X 0,Y 140.616,Z 784.64,A -85,B 0,C 180,E1 -24204.259,E2 -24204.259} C_VEL
LIN {X 0,Y 140.559,Z 785.226,A -85,B 0,C 180,E1 -24209.996,E2 -24209.996} C_VEL
LIN {X 0,Y 140.614,Z 784.624,A -85,B 0,C 180,E1 -24215.732,E2 -24215.732} C_VEL
LIN {X 0,Y 141.351,Z 782.874,A -85,B 0,C 180,E1 -24221.467,E2 -24221.467} C_VEL
LIN {X 0,Y 143.039,Z 779.948,A -85,B 0,C 180,E1 -24227.141,E2 -24227.141} C_VEL
LIN {X 0,Y 145.965,Z 775.774,A -85,B 0,C 180,E1 -24232.65,E2 -24232.65} C_VEL
LIN {X 0,Y 149.983,Z 770.24,A -85,B 0,C 180,E1 -24237.937,E2 -24237.937} C_VEL
LIN {X 0,Y 155.192,Z 763.195,A -85,B 0,C 180,E1 -24242.912,E2 -24242.912} C_VEL
LIN {X 0,Y 160.677,Z 755.644,A -85,B 0,C 180,E1 -24246.966,E2 -24246.966} C_VEL
LIN {X 0,Y 166.619,Z 746.546,A -85,B 0,C 180,E1 -24250.821,E2 -24250.821} C_VEL
LIN {X 0,Y 172.503,Z 737.267,A -85,B 0,C 180,E1 -24253.831,E2 -24253.831} C_VEL
LIN {X 0,Y 179.296,Z 725.239,A -85,B 0,C 180,E1 -24256.885,E2 -24256.885} C_VEL
LIN {X 0,Y 185.442,Z 712.954,A -85,B 0,C 180,E1 -24259.28,E2 -24259.28} C_VEL
LIN {X 0,Y 191.106,Z 699.674,A -85,B 0,C 180,E1 -24261.305,E2 -24261.305} C_VEL
LIN {X 0,Y 196.007,Z 686.008,A -85,B 0,C 180,E1 -24262.913,E2 -24262.913} C_VEL
LIN {X 0,Y 200.35,Z 671.206,A -85,B 0,C 180,E1 -24264.206,E2 -24264.206} C_VEL
LIN {X 0,Y 203.708,Z 656.458,A -85,B 0,C 180,E1 -24265.125,E2 -24265.125} C_VEL
LIN {X 0,Y 206.071,Z 641.248,A -85,B 0,C 180,E1 -24265.789,E2 -24265.789} C_VEL
LIN {X 0,Y 212.664,Z 563.302,A -85,B 0,C 180,E1 -24267.915,E2 -24267.915} C_VEL
LIN {X 0,Y 215.281,Z 530.859,A -85,B 0,C 180,E1 -24268.811,E2 -24268.811} C_VEL
LIN {X 0,Y 214.982,Z 515.342,A -85,B 0,C 180,E1 -24269.945,E2 -24269.945} C_VEL
LIN {X 0,Y 213.418,Z 509.554,A -85,B 0,C 180,E1 -24271.075,E2 -24271.075} C_VEL
LIN {X 0,Y 209.307,Z 502.598,A -85,B 0,C 180,E1 -24273.717,E2 -24273.717} C_VEL
LIN {X 0,Y 205.15,Z 496.305,A -85,B 0,C 180,E1 -24276.732,E2 -24276.732} C_VEL
LIN {X 0,Y 201.095,Z 490.362,A -85,B 0,C 180,E1 -24280.211,E2 -24280.211} C_VEL
LIN {X 0,Y 198.195,Z 486.527,A -85,B 0,C 180,E1 -24283.175,E2 -24283.175} C_VEL
LIN {X 0,Y 194.109,Z 481.252,A -85,B 0,C 180,E1 -24288.778,E2 -24288.778} C_VEL
LIN {X 0,Y 192.271,Z 479.078,A -85,B 0,C 180,E1 -24292.65,E2 -24292.65} C_VEL
LIN {X 0,Y 190.99,Z 477.983,A -85,B 0,C 180,E1 -24297.891,E2 -24297.891} C_VEL
LIN {X 0,Y 190.921,Z 478.282,A -85,B 0,C 180,E1 -24301.582,E2 -24301.582} C_VEL
LIN {X 0,Y 191.573,Z 479.909,A -85,B 0,C 180,E1 -24305.551,E2 -24305.551} C_VEL
LIN {X 0,Y 193.598,Z 483.886,A -85,B 0,C 180,E1 -24310.722,E2 -24310.722} C_VEL
LIN {X 0,Y 196.87,Z 489.541,A -85,B 0,C 180,E1 -24315.665,E2 -24315.665} C_VEL
LIN {X 0,Y 200.33,Z 495.928,A -85,B 0,C 180,E1 -24319.534,E2 -24319.534} C_VEL
LIN {X 0,Y 203.733,Z 502.302,A -85,B 0,C 180,E1 -24322.636,E2 -24322.636} C_VEL
LIN {X 0,Y 207.387,Z 509.837,A -85,B 0,C 180,E1 -24325.532,E2 -24325.532} C_VEL
LIN {X 0,Y 211.346,Z 518.806,A -85,B 0,C 180,E1 -24328.319,E2 -24328.319} C_VEL
LIN {X 0,Y 214.761,Z 527.369,A -85,B 0,C 180,E1 -24330.514,E2 -24330.514} C_VEL
LIN {X 0,Y 215.088,Z 539.065,A -85,B 0,C 180,E1 -24331.402,E2 -24331.402} C_VEL
LIN {X 0,Y 206.615,Z 639.587,A -85,B 0,C 180,E1 -24334.107,E2 -24334.107} C_VEL
LIN {X 0,Y 204.427,Z 654.566,A -85,B 0,C 180,E1 -24334.734,E2 -24334.734} C_VEL
LIN {X 0,Y 201.419,Z 668.618,A -85,B 0,C 180,E1 -24335.574,E2 -24335.574} C_VEL
LIN {X 0,Y 197.308,Z 683.082,A -85,B 0,C 180,E1 -24336.739,E2 -24336.739} C_VEL
LIN {X 0,Y 192.348,Z 697.411,A -85,B 0,C 180,E1 -24338.329,E2 -24338.329} C_VEL
LIN {X 0,Y 186.696,Z 711.118,A -85,B 0,C 180,E1 -24340.339,E2 -24340.339} C_VEL
LIN {X 0,Y 180.424,Z 723.769,A -85,B 0,C 180,E1 -24342.679,E2 -24342.679} C_VEL
LIN {X 0,Y 174.597,Z 734.362,A -85,B 0,C 180,E1 -24345.223,E2 -24345.223} C_VEL
LIN {X 0,Y 168.618,Z 744.164,A -85,B 0,C 180,E1 -24348.179,E2 -24348.179} C_VEL
LIN {X 0,Y 163.288,Z 752.518,A -85,B 0,C 180,E1 -24351.39,E2 -24351.39} C_VEL
LIN {X 0,Y 157.431,Z 760.68,A -85,B 0,C 180,E1 -24355.312,E2 -24355.312} C_VEL
LIN {X 0,Y 152.505,Z 767.44,A -85,B 0,C 180,E1 -24359.546,E2 -24359.546} C_VEL
LIN {X 0,Y 147.911,Z 773.704,A -85,B 0,C 180,E1 -24364.687,E2 -24364.687} C_VEL
LIN {X 0,Y 144.429,Z 778.543,A -85,B 0,C 180,E1 -24370.09,E2 -24370.09} C_VEL
LIN {X 0,Y 142.016,Z 782.088,A -85,B 0,C 180,E1 -24375.679,E2 -24375.679} C_VEL
LIN {X 0,Y 140.77,Z 784.428,A -85,B 0,C 180,E1 -24381.391,E2 -24381.391} C_VEL
LIN {X 0,Y 140.429,Z 785.616,A -85,B 0,C 180,E1 -24387.136,E2 -24387.136} C_VEL
LIN {X 0,Y 140.486,Z 785.773,A -85,B 0,C 180,E1 -24390.004,E2 -24390.004} C_VEL
LIN {X 0,Y 140.534,Z 785.195,A -85,B 0,C 180,E1 -24395.745,E2 -24395.745} C_VEL
LIN {X 0,Y 141.291,Z 783.475,A -85,B 0,C 180,E1 -24401.481,E2 -24401.481} C_VEL
LIN {X 0,Y 143.003,Z 780.577,A -85,B 0,C 180,E1 -24407.154,E2 -24407.154} C_VEL
LIN {X 0,Y 145.965,Z 776.434,A -85,B 0,C 180,E1 -24412.66,E2 -24412.66} C_VEL
LIN {X 0,Y 149.985,Z 770.946,A -85,B 0,C 180,E1 -24417.947,E2 -24417.947} C_VEL
LIN {X 0,Y 155.158,Z 763.96,A -85,B 0,C 180,E1 -24422.93,E2 -24422.93} C_VEL
LIN {X 0,Y 160.647,Z 756.469,A -85,B 0,C 180,E1 -24426.984,E2 -24426.984} C_VEL
LIN {X 0,Y 166.673,Z 747.443,A -85,B 0,C 180,E1 -24430.815,E2 -24430.815} C_VEL
LIN {X 0,Y 172.492,Z 738.226,A -85,B 0,C 180,E1 -24433.844,E2 -24433.844} C_VEL
LIN {X 0,Y 179.256,Z 726.343,A -85,B 0,C 180,E1 -24436.909,E2 -24436.909} C_VEL
LIN {X 0,Y 185.447,Z 714.214,A -85,B 0,C 180,E1 -24439.288,E2 -24439.288} C_VEL
LIN {X 0,Y 190.877,Z 701.685,A -85,B 0,C 180,E1 -24441.249,E2 -24441.249} C_VEL
LIN {X 0,Y 195.989,Z 687.796,A -85,B 0,C 180,E1 -24442.931,E2 -24442.931} C_VEL
LIN {X 0,Y 200.34,Z 673.464,A -85,B 0,C 180,E1 -24444.221,E2 -24444.221} C_VEL
LIN {X 0,Y 204.011,Z 657.881,A -85,B 0,C 180,E1 -24445.229,E2 -24445.229} C_VEL
LIN {X 0,Y 206.467,Z 642.578,A -85,B 0,C 180,E1 -24445.928,E2 -24445.928} C_VEL
LIN {X 0,Y 207.656,Z 630.199,A -85,B 0,C 180,E1 -24446.322,E2 -24446.322} C_VEL
LIN {X 0,Y 203.099,Z 636.649,A -85,B 0,C 180,E1 -24447.84,E2 -24447.84} C_VEL
LIN {X 0,Y 199.913,Z 640.396,A -85,B 0,C 180,E1 -24448.986,E2 -24448.986} C_VEL
LIN {X 0,Y 193.796,Z 650.212,A -85,B 0,C 180,E1 -24450.96,E2 -24450.96} C_VEL
LIN {X 0,Y 187.755,Z 657.876,A -85,B 0,C 180,E1 -24453.143,E2 -24453.143} C_VEL
LIN {X 0,Y 182.905,Z 662.652,A -85,B 0,C 180,E1 -24455.224,E2 -24455.224} C_VEL
LIN {X 0,Y 181.364,Z 663.96,A -85,B 0,C 180,E1 -24455.991,E2 -24455.991} C_VEL
LIN {X 0,Y 175.868,Z 670.62,A -85,B 0,C 180,E1 -24458.306,E2 -24458.306} C_VEL
LIN {X 0,Y 172.676,Z 674.054,A -85,B 0,C 180,E1 -24459.884,E2 -24459.884} C_VEL
LIN {X 0,Y 169.35,Z 677.028,A -85,B 0,C 180,E1 -24461.865,E2 -24461.865} C_VEL
LIN {X 0,Y 166.42,Z 679.28,A -85,B 0,C 180,E1 -24464.068,E2 -24464.068} C_VEL
LIN {X 0,Y 161.507,Z 684.591,A -85,B 0,C 180,E1 -24467.433,E2 -24467.433} C_VEL
LIN {X 0,Y 158.987,Z 687.097,A -85,B 0,C 180,E1 -24469.815,E2 -24469.815} C_VEL
LIN {X 0,Y 155.107,Z 691.011,A -85,B 0,C 180,E1 -24474.8,E2 -24474.8} C_VEL
LIN {X 0,Y 153.328,Z 693.541,A -85,B 0,C 180,E1 -24477.373,E2 -24477.373} C_VEL
LIN {X 0,Y 152.218,Z 695.236,A -85,B 0,C 180,E1 -24480,E2 -24480} C_VEL
LIN {X 0,Y 151.331,Z 697.904,A -85,B 0,C 180,E1 -24485.329,E2 -24485.329} C_VEL
LIN {X 0,Y 151.13,Z 699.699,A -85,B 0,C 180,E1 -24488.019,E2 -24488.019} C_VEL
LIN {X 0,Y 151.473,Z 701.048,A -85,B 0,C 180,E1 -24490.695,E2 -24490.695} C_VEL
LIN {X 0,Y 154.146,Z 703.015,A -85,B 0,C 180,E1 -24496.761,E2 -24496.761} C_VEL
LIN {X 0,Y 156.899,Z 704.74,A -85,B 0,C 180,E1 -24500.998,E2 -24500.998} C_VEL
LIN {X 0,Y 161.963,Z 705.583,A -85,B 0,C 180,E1 -24505.717,E2 -24505.717} C_VEL
LIN {X 0,Y 167.008,Z 705.933,A -85,B 0,C 180,E1 -24508.943,E2 -24508.943} C_VEL
LIN {X 0,Y 177.052,Z 707.522,A -85,B 0,C 180,E1 -24513.76,E2 -24513.76} C_VEL
LIN {X 0,Y 186.203,Z 707.707,A -85,B 0,C 180,E1 -24517.149,E2 -24517.149} C_VEL
LIN {X 0,Y 191.046,Z 707.424,A -85,B 0,C 180,E1 -24518.71,E2 -24518.71} C_VEL
LIN {X 0,Y 190.46,Z 707.856,A -85,B 0,C 180,E1 -24519.2,E2 -24519.2} C_VEL
LIN {X 0,Y 187.371,Z 709.293,A -85,B 0,C 180,E1 -24520.053,E2 -24520.053} C_VEL
LIN {X 0,Y 183.904,Z 716.513,A -85,B 0,C 180,E1 -24521.319,E2 -24521.319} C_VEL
LIN {X 0,Y 181.083,Z 721.209,A -85,B 0,C 180,E1 -24522.048,E2 -24522.048} C_VEL
LIN {X 0,Y 175.15,Z 728.586,A -85,B 0,C 180,E1 -24522.989,E2 -24522.989} C_VEL
LIN {X 0,Y 169.057,Z 735.643,A -85,B 0,C 180,E1 -24524.118,E2 -24524.118} C_VEL
LIN {X 0,Y 166.035,Z 739.68,A -85,B 0,C 180,E1 -24525.152,E2 -24525.152} C_VEL
LIN {X 0,Y 159.475,Z 749.472,A -85,B 0,C 180,E1 -24528.616,E2 -24528.616} C_VEL
LIN {X 0,Y 153.342,Z 758.087,A -85,B 0,C 180,E1 -24532.603,E2 -24532.603} C_VEL
LIN {X 0,Y 147.801,Z 765.247,A -85,B 0,C 180,E1 -24536.846,E2 -24536.846} C_VEL
LIN {X 0,Y 142.555,Z 771.867,A -85,B 0,C 180,E1 -24542.068,E2 -24542.068} C_VEL
LIN {X 0,Y 138.51,Z 777.039,A -85,B 0,C 180,E1 -24547.628,E2 -24547.628} C_VEL
LIN {X 0,Y 136.241,Z 780.015,A -85,B 0,C 180,E1 -24551.966,E2 -24551.966} C_VEL
LIN {X 0,Y 134.36,Z 782.925,A -85,B 0,C 180,E1 -24557.918,E2 -24557.918} C_VEL
LIN {X 0,Y 133.541,Z 784.654,A -85,B 0,C 180,E1 -24563.953,E2 -24563.953} C_VEL
LIN {X 0,Y 133.456,Z 785.239,A -85,B 0,C 180,E1 -24569.995,E2 -24569.995} C_VEL
LIN {X 0,Y 133.539,Z 784.638,A -85,B 0,C 180,E1 -24576.037,E2 -24576.037} C_VEL
LIN {X 0,Y 134.35,Z 782.888,A -85,B 0,C 180,E1 -24582.073,E2 -24582.073} C_VEL
LIN {X 0,Y 136.224,Z 779.962,A -85,B 0,C 180,E1 -24588.027,E2 -24588.027} C_VEL
LIN {X 0,Y 139.395,Z 775.788,A -85,B 0,C 180,E1 -24593.782,E2 -24593.782} C_VEL
LIN {X 0,Y 143.698,Z 770.254,A -85,B 0,C 180,E1 -24599.275,E2 -24599.275} C_VEL
LIN {X 0,Y 149.227,Z 763.209,A -85,B 0,C 180,E1 -24604.407,E2 -24604.407} C_VEL
LIN {X 0,Y 155.011,Z 755.659,A -85,B 0,C 180,E1 -24608.56,E2 -24608.56} C_VEL
LIN {X 0,Y 161.284,Z 746.559,A -85,B 0,C 180,E1 -24612.481,E2 -24612.481} C_VEL
LIN {X 0,Y 167.427,Z 737.284,A -85,B 0,C 180,E1 -24615.523,E2 -24615.523} C_VEL
LIN {X 0,Y 174.515,Z 725.258,A -85,B 0,C 180,E1 -24618.589,E2 -24618.589} C_VEL
LIN {X 0,Y 180.883,Z 712.975,A -85,B 0,C 180,E1 -24620.987,E2 -24620.987} C_VEL
LIN {X 0,Y 186.747,Z 699.698,A -85,B 0,C 180,E1 -24623.006,E2 -24623.006} C_VEL
LIN {X 0,Y 191.812,Z 686.037,A -85,B 0,C 180,E1 -24624.604,E2 -24624.604} C_VEL
LIN {X 0,Y 196.291,Z 671.242,A -85,B 0,C 180,E1 -24625.884,E2 -24625.884} C_VEL
LIN {X 0,Y 199.738,Z 656.508,A -85,B 0,C 180,E1 -24626.794,E2 -24626.794} C_VEL
LIN {X 0,Y 202.168,Z 641.328,A -85,B 0,C 180,E1 -24627.452,E2 -24627.452} C_VEL
LIN {X 0,Y 209.143,Z 561.561,A -85,B 0,C 180,E1 -24629.612,E2 -24629.612} C_VEL
LIN {X 0,Y 211.627,Z 531.97,A -85,B 0,C 180,E1 -24630.419,E2 -24630.419} C_VEL
LIN {X 0,Y 211.464,Z 518.427,A -85,B 0,C 180,E1 -24631.428,E2 -24631.428} C_VEL
LIN {X 0,Y 210.395,Z 514.464,A -85,B 0,C 180,E1 -24632.253,E2 -24632.253} C_VEL
LIN {X 0,Y 206.785,Z 508.203,A -85,B 0,C 180,E1 -24634.725,E2 -24634.725} C_VEL
LIN {X 0,Y 202.38,Z 501.271,A -85,B 0,C 180,E1 -24638.169,E2 -24638.169} C_VEL
LIN {X 0,Y 198.163,Z 495.007,A -85,B 0,C 180,E1 -24642.188,E2 -24642.188} C_VEL
LIN {X 0,Y 193.769,Z 489.215,A -85,B 0,C 180,E1 -24647.83,E2 -24647.83} C_VEL
LIN {X 0,Y 191.719,Z 486.503,A -85,B 0,C 180,E1 -24651.834,E2 -24651.834} C_VEL
LIN {X 0,Y 190.456,Z 485.398,A -85,B 0,C 180,E1 -24655.768,E2 -24655.768} C_VEL
LIN {X 0,Y 190.011,Z 485.018,A -85,B 0,C 180,E1 -24660,E2 -24660} C_VEL
LIN {X 0,Y 190.394,Z 486.362,A -85,B 0,C 180,E1 -24664.234,E2 -24664.234} C_VEL
LIN {X 0,Y 191.966,Z 489.747,A -85,B 0,C 180,E1 -24669.217,E2 -24669.217} C_VEL
LIN {X 0,Y 195.024,Z 495.375,A -85,B 0,C 180,E1 -24674.478,E2 -24674.478} C_VEL
LIN {X 0,Y 198.406,Z 501.935,A -85,B 0,C 180,E1 -24678.591,E2 -24678.591} C_VEL
LIN {X 0,Y 201.744,Z 508.56,A -85,B 0,C 180,E1 -24681.842,E2 -24681.842} C_VEL
LIN {X 0,Y 204.906,Z 515.363,A -85,B 0,C 180,E1 -24684.507,E2 -24684.507} C_VEL
LIN {X 0,Y 208.564,Z 524.101,A -85,B 0,C 180,E1 -24687.265,E2 -24687.265} C_VEL
LIN {X 0,Y 211.195,Z 530.919,A -85,B 0,C 180,E1 -24689.082,E2 -24689.082} C_VEL
LIN {X 0,Y 211.345,Z 540.42,A -85,B 0,C 180,E1 -24689.796,E2 -24689.796} C_VEL
LIN {X 0,Y 202.72,Z 639.51,A -85,B 0,C 180,E1 -24692.446,E2 -24692.446} C_VEL
LIN {X 0,Y 200.475,Z 654.517,A -85,B 0,C 180,E1 -24693.07,E2 -24693.07} C_VEL
LIN {X 0,Y 197.379,Z 668.583,A -85,B 0,C 180,E1 -24693.9,E2 -24693.9} C_VEL
LIN {X 0,Y 193.143,Z 683.053,A -85,B 0,C 180,E1 -24695.05,E2 -24695.05} C_VEL
LIN {X 0,Y 188.161,Z 697.043,A -85,B 0,C 180,E1 -24696.586,E2 -24696.586} C_VEL
LIN {X 0,Y 182.785,Z 709.826,A -85,B 0,C 180,E1 -24698.433,E2 -24698.433} C_VEL
LIN {X 0,Y 176.871,Z 721.643,A -85,B 0,C 180,E1 -24700.548,E2 -24700.548} C_VEL
LIN {X 0,Y 170.67,Z 732.585,A -85,B 0,C 180,E1 -24703.042,E2 -24703.042} C_VEL
LIN {X 0,Y 164.366,Z 742.662,A -85,B 0,C 180,E1 -24705.993,E2 -24705.993} C_VEL
LIN {X 0,Y 157.741,Z 752.503,A -85,B 0,C 180,E1 -24709.763,E2 -24709.763} C_VEL
LIN {X 0,Y 151.603,Z 760.665,A -85,B 0,C 180,E1 -24713.773,E2 -24713.773} C_VEL
LIN {X 0,Y 146.383,Z 767.425,A -85,B 0,C 180,E1 -24718.127,E2 -24718.127} C_VEL
LIN {X 0,Y 141.467,Z 773.69,A -85,B 0,C 180,E1 -24723.447,E2 -24723.447} C_VEL
LIN {X 0,Y 137.732,Z 778.53,A -85,B 0,C 180,E1 -24729.078,E2 -24729.078} C_VEL
LIN {X 0,Y 135.108,Z 782.074,A -85,B 0,C 180,E1 -24734.93,E2 -24734.93} C_VEL
LIN {X 0,Y 133.727,Z 784.415,A -85,B 0,C 180,E1 -24740.933,E2 -24740.933} C_VEL
LIN {X 0,Y 133.331,Z 785.603,A -85,B 0,C 180,E1 -24746.983,E2 -24746.983} C_VEL
LIN {X 0,Y 133.392,Z 785.76,A -85,B 0,C 180,E1 -24750.005,E2 -24750.005} C_VEL
LIN {X 0,Y 133.451,Z 785.181,A -85,B 0,C 180,E1 -24756.051,E2 -24756.051} C_VEL
LIN {X 0,Y 134.297,Z 783.461,A -85,B 0,C 180,E1 -24762.088,E2 -24762.088} C_VEL
LIN {X 0,Y 136.193,Z 780.562,A -85,B 0,C 180,E1 -24768.041,E2 -24768.041} C_VEL
LIN {X 0,Y 139.392,Z 776.418,A -85,B 0,C 180,E1 -24773.793,E2 -24773.793} C_VEL
LIN {X 0,Y 143.702,Z 770.929,A -85,B 0,C 180,E1 -24779.284,E2 -24779.284} C_VEL
LIN {X 0,Y 149.183,Z 763.942,A -85,B 0,C 180,E1 -24784.429,E2 -24784.429} C_VEL
LIN {X 0,Y 155,Z 756.45,A -85,B 0,C 180,E1 -24788.573,E2 -24788.573} C_VEL
LIN {X 0,Y 161.336,Z 747.423,A -85,B 0,C 180,E1 -24792.472,E2 -24792.472} C_VEL
LIN {X 0,Y 167.406,Z 738.204,A -85,B 0,C 180,E1 -24795.541,E2 -24795.541} C_VEL
LIN {X 0,Y 174.461,Z 726.318,A -85,B 0,C 180,E1 -24798.62,E2 -24798.62} C_VEL
LIN {X 0,Y 180.878,Z 714.186,A -85,B 0,C 180,E1 -24801,E2 -24801} C_VEL
LIN {X 0,Y 186.616,Z 701.396,A -85,B 0,C 180,E1 -24802.991,E2 -24802.991} C_VEL
LIN {X 0,Y 191.786,Z 687.757,A -85,B 0,C 180,E1 -24804.627,E2 -24804.627} C_VEL
LIN {X 0,Y 196.058,Z 674.153,A -85,B 0,C 180,E1 -24805.842,E2 -24805.842} C_VEL
LIN {X 0,Y 199.857,Z 658.748,A -85,B 0,C 180,E1 -24806.846,E2 -24806.846} C_VEL
LIN {X 0,Y 202.181,Z 644.916,A -85,B 0,C 180,E1 -24807.516,E2 -24807.516} C_VEL
LIN {X 0,Y 194.865,Z 655.613,A -85,B 0,C 180,E1 -24809.62,E2 -24809.62} C_VEL
LIN {X 0,Y 188.225,Z 663.39,A -85,B 0,C 180,E1 -24811.799,E2 -24811.799} C_VEL
LIN {X 0,Y 183.086,Z 668.238,A -85,B 0,C 180,E1 -24813.804,E2 -24813.804} C_VEL
LIN {X 0,Y 180.999,Z 670.001,A -85,B 0,C 180,E1 -24814.715,E2 -24814.715} C_VEL
LIN {X 0,Y 175.301,Z 676.281,A -85,B 0,C 180,E1 -24816.927,E2 -24816.927} C_VEL
LIN {X 0,Y 170.842,Z 680.591,A -85,B 0,C 180,E1 -24819.018,E2 -24819.018} C_VEL
LIN {X 0,Y 166.539,Z 683.94,A -85,B 0,C 180,E1 -24821.548,E2 -24821.548} C_VEL
LIN {X 0,Y 164.974,Z 685.049,A -85,B 0,C 180,E1 -24822.65,E2 -24822.65} C_VEL
LIN {X 0,Y 158.99,Z 690.823,A -85,B 0,C 180,E1 -24826.543,E2 -24826.543} C_VEL
LIN {X 0,Y 155.715,Z 693.671,A -85,B 0,C 180,E1 -24829.599,E2 -24829.599} C_VEL
LIN {X 0,Y 152.513,Z 696.562,A -85,B 0,C 180,E1 -24833.45,E2 -24833.45} C_VEL
LIN {X 0,Y 150.491,Z 699,A -85,B 0,C 180,E1 -24835.983,E2 -24835.983} C_VEL
LIN {X 0,Y 148.631,Z 701.511,A -85,B 0,C 180,E1 -24840,E2 -24840} C_VEL
LIN {X 0,Y 147.557,Z 704.251,A -85,B 0,C 180,E1 -24845.466,E2 -24845.466} C_VEL
LIN {X 0,Y 147.367,Z 705.88,A -85,B 0,C 180,E1 -24848.225,E2 -24848.225} C_VEL
LIN {X 0,Y 147.744,Z 707.115,A -85,B 0,C 180,E1 -24850.969,E2 -24850.969} C_VEL
LIN {X 0,Y 149.969,Z 708.712,A -85,B 0,C 180,E1 -24856.33,E2 -24856.33} C_VEL
LIN {X 0,Y 153.222,Z 710.663,A -85,B 0,C 180,E1 -24861.527,E2 -24861.527} C_VEL
LIN {X 0,Y 158.393,Z 711.457,A -85,B 0,C 180,E1 -24866.34,E2 -24866.34} C_VEL
LIN {X 0,Y 164.918,Z 711.739,A -85,B 0,C 180,E1 -24870.756,E2 -24870.756} C_VEL
LIN {X 0,Y 172.421,Z 711.882,A -85,B 0,C 180,E1 -24874.795,E2 -24874.795} C_VEL
LIN {X 0,Y 181.243,Z 711.046,A -85,B 0,C 180,E1 -24878.347,E2 -24878.347} C_VEL
LIN {X 0,Y 181.277,Z 712.579,A -85,B 0,C 180,E1 -24878.908,E2 -24878.908} C_VEL
LIN {X 0,Y 174.554,Z 725.51,A -85,B 0,C 180,E1 -24881.414,E2 -24881.414} C_VEL
LIN {X 0,Y 167.467,Z 737.483,A -85,B 0,C 180,E1 -24884.481,E2 -24884.481} C_VEL
LIN {X 0,Y 166.035,Z 739.68,A -85,B 0,C 180,E1 -24885.152,E2 -24885.152} C_VEL
LIN {X 0,Y 163.001,Z 743.626,A -85,B 0,C 180,E1 -24886.272,E2 -24886.272} C_VEL
LIN {X 0,Y 156.707,Z 749.763,A -85,B 0,C 180,E1 -24887.9,E2 -24887.9} C_VEL
LIN {X 0,Y 150.333,Z 755.504,A -85,B 0,C 180,E1 -24889.759,E2 -24889.759} C_VEL
LIN {X 0,Y 147.243,Z 758.709,A -85,B 0,C 180,E1 -24891.245,E2 -24891.245} C_VEL
LIN {X 0,Y 141.859,Z 765.265,A -85,B 0,C 180,E1 -24895.264,E2 -24895.264} C_VEL
LIN {X 0,Y 136.28,Z 771.883,A -85,B 0,C 180,E1 -24900.66,E2 -24900.66} C_VEL
LIN {X 0,Y 131.91,Z 777.054,A -85,B 0,C 180,E1 -24906.443,E2 -24906.443} C_VEL
LIN {X 0,Y 129.467,Z 780.03,A -85,B 0,C 180,E1 -24910.987,E2 -24910.987} C_VEL
LIN {X 0,Y 127.388,Z 782.94,A -85,B 0,C 180,E1 -24917.246,E2 -24917.246} C_VEL
LIN {X 0,Y 126.462,Z 784.668,A -85,B 0,C 180,E1 -24923.614,E2 -24923.614} C_VEL
LIN {X 0,Y 126.362,Z 785.253,A -85,B 0,C 180,E1 -24929.995,E2 -24929.995} C_VEL
LIN {X 0,Y 126.459,Z 784.652,A -85,B 0,C 180,E1 -24936.377,E2 -24936.377} C_VEL
LIN {X 0,Y 127.377,Z 782.901,A -85,B 0,C 180,E1 -24942.745,E2 -24942.745} C_VEL
LIN {X 0,Y 129.451,Z 779.975,A -85,B 0,C 180,E1 -24949.005,E2 -24949.005} C_VEL
LIN {X 0,Y 132.883,Z 775.801,A -85,B 0,C 180,E1 -24955.025,E2 -24955.025} C_VEL
LIN {X 0,Y 137.501,Z 770.268,A -85,B 0,C 180,E1 -24960.733,E2 -24960.733} C_VEL
LIN {X 0,Y 143.359,Z 763.224,A -85,B 0,C 180,E1 -24966.029,E2 -24966.029} C_VEL
LIN {X 0,Y 149.483,Z 755.674,A -85,B 0,C 180,E1 -24970.269,E2 -24970.269} C_VEL
LIN {X 0,Y 155.072,Z 747.983,A -85,B 0,C 180,E1 -24973.714,E2 -24973.714} C_VEL
LIN {X 0,Y 162.517,Z 737.301,A -85,B 0,C 180,E1 -24977.314,E2 -24977.314} C_VEL
LIN {X 0,Y 169.891,Z 725.277,A -85,B 0,C 180,E1 -24980.39,E2 -24980.39} C_VEL
LIN {X 0,Y 176.488,Z 712.996,A -85,B 0,C 180,E1 -24982.783,E2 -24982.783} C_VEL
LIN {X 0,Y 182.558,Z 699.723,A -85,B 0,C 180,E1 -24984.788,E2 -24984.788} C_VEL
LIN {X 0,Y 187.782,Z 686.066,A -85,B 0,C 180,E1 -24986.374,E2 -24986.374} C_VEL
LIN {X 0,Y 192.396,Z 671.279,A -85,B 0,C 180,E1 -24987.636,E2 -24987.636} C_VEL
LIN {X 0,Y 195.944,Z 656.559,A -85,B 0,C 180,E1 -24988.529,E2 -24988.529} C_VEL
LIN {X 0,Y 198.446,Z 641.408,A -85,B 0,C 180,E1 -24989.177,E2 -24989.177} C_VEL
LIN {X 0,Y 205.585,Z 562.428,A -85,B 0,C 180,E1 -24991.294,E2 -24991.294} C_VEL
LIN {X 0,Y 208.147,Z 532.717,A -85,B 0,C 180,E1 -24992.107,E2 -24992.107} C_VEL
LIN {X 0,Y 208.112,Z 521.563,A -85,B 0,C 180,E1 -24992.945,E2 -24992.945} C_VEL
LIN {X 0,Y 207.545,Z 519.529,A -85,B 0,C 180,E1 -24993.409,E2 -24993.409} C_VEL
LIN {X 0,Y 204.027,Z 513.314,A -85,B 0,C 180,E1 -24995.99,E2 -24995.99} C_VEL
LIN {X 0,Y 199.043,Z 505.235,A -85,B 0,C 180,E1 -25000.303,E2 -25000.303} C_VEL
LIN {X 0,Y 195.862,Z 500.545,A -85,B 0,C 180,E1 -25003.708,E2 -25003.708} C_VEL
LIN {X 0,Y 192.085,Z 495.296,A -85,B 0,C 180,E1 -25009.193,E2 -25009.193} C_VEL
LIN {X 0,Y 190.551,Z 493.21,A -85,B 0,C 180,E1 -25012.583,E2 -25012.583} C_VEL
LIN {X 0,Y 189.26,Z 492.095,A -85,B 0,C 180,E1 -25017.872,E2 -25017.872} C_VEL
LIN {X 0,Y 189.16,Z 492.281,A -85,B 0,C 180,E1 -25021.065,E2 -25021.065} C_VEL
LIN {X 0,Y 189.662,Z 493.827,A -85,B 0,C 180,E1 -25024.929,E2 -25024.929} C_VEL
LIN {X 0,Y 191.252,Z 497.443,A -85,B 0,C 180,E1 -25029.652,E2 -25029.652} C_VEL
LIN {X 0,Y 193.871,Z 502.525,A -85,B 0,C 180,E1 -25034.197,E2 -25034.197} C_VEL
LIN {X 0,Y 196.75,Z 508.406,A -85,B 0,C 180,E1 -25037.875,E2 -25037.875} C_VEL
LIN {X 0,Y 199.706,Z 514.59,A -85,B 0,C 180,E1 -25040.942,E2 -25040.942} C_VEL
LIN {X 0,Y 202.584,Z 521.16,A -85,B 0,C 180,E1 -25043.54,E2 -25043.54} C_VEL
LIN {X 0,Y 206.22,Z 530.291,A -85,B 0,C 180,E1 -25046.456,E2 -25046.456} C_VEL
LIN {X 0,Y 207.787,Z 534.56,A -85,B 0,C 180,E1 -25047.62,E2 -25047.62} C_VEL
LIN {X 0,Y 207.817,Z 541.309,A -85,B 0,C 180,E1 -25048.123,E2 -25048.123} C_VEL
LIN {X 0,Y 198.848,Z 640.828,A -85,B 0,C 180,E1 -25050.77,E2 -25050.77} C_VEL
LIN {X 0,Y 196.361,Z 656.219,A -85,B 0,C 180,E1 -25051.424,E2 -25051.424} C_VEL
LIN {X 0,Y 192.836,Z 671.065,A -85,B 0,C 180,E1 -25052.327,E2 -25052.327} C_VEL
LIN {X 0,Y 188.499,Z 684.963,A -85,B 0,C 180,E1 -25053.471,E2 -25053.471} C_VEL
LIN {X 0,Y 183.582,Z 698.064,A -85,B 0,C 180,E1 -25054.939,E2 -25054.939} C_VEL
LIN {X 0,Y 177.79,Z 711.128,A -85,B 0,C 180,E1 -25056.85,E2 -25056.85} C_VEL
LIN {X 0,Y 171.105,Z 723.732,A -85,B 0,C 180,E1 -25059.177,E2 -25059.177} C_VEL
LIN {X 0,Y 164.752,Z 734.327,A -85,B 0,C 180,E1 -25061.717,E2 -25061.717} C_VEL
LIN {X 0,Y 158.254,Z 744.132,A -85,B 0,C 180,E1 -25064.727,E2 -25064.727} C_VEL
LIN {X 0,Y 152.239,Z 752.619,A -85,B 0,C 180,E1 -25068.079,E2 -25068.079} C_VEL
LIN {X 0,Y 145.909,Z 760.65,A -85,B 0,C 180,E1 -25072.117,E2 -25072.117} C_VEL
LIN {X 0,Y 140.344,Z 767.411,A -85,B 0,C 180,E1 -25076.581,E2 -25076.581} C_VEL
LIN {X 0,Y 134.902,Z 773.918,A -85,B 0,C 180,E1 -25082.333,E2 -25082.333} C_VEL
LIN {X 0,Y 131.081,Z 778.516,A -85,B 0,C 180,E1 -25087.962,E2 -25087.962} C_VEL
LIN {X 0,Y 128.209,Z 782.06,A -85,B 0,C 180,E1 -25094.098,E2 -25094.098} C_VEL
LIN {X 0,Y 126.705,Z 784.401,A -85,B 0,C 180,E1 -25100.426,E2 -25100.426} C_VEL
LIN {X 0,Y 126.244,Z 785.589,A -85,B 0,C 180,E1 -25106.814,E2 -25106.814} C_VEL
LIN {X 0,Y 126.308,Z 785.746,A -85,B 0,C 180,E1 -25110.005,E2 -25110.005} C_VEL
LIN {X 0,Y 126.374,Z 785.167,A -85,B 0,C 180,E1 -25116.391,E2 -25116.391} C_VEL
LIN {X 0,Y 127.331,Z 783.446,A -85,B 0,C 180,E1 -25122.76,E2 -25122.76} C_VEL
LIN {X 0,Y 129.425,Z 780.547,A -85,B 0,C 180,E1 -25129.019,E2 -25129.019} C_VEL
LIN {X 0,Y 132.881,Z 776.402,A -85,B 0,C 180,E1 -25135.036,E2 -25135.036} C_VEL
LIN {X 0,Y 137.5,Z 770.913,A -85,B 0,C 180,E1 -25140.744,E2 -25140.744} C_VEL
LIN {X 0,Y 143.328,Z 763.924,A -85,B 0,C 180,E1 -25146.049,E2 -25146.049} C_VEL
LIN {X 0,Y 149.481,Z 756.431,A -85,B 0,C 180,E1 -25150.281,E2 -25150.281} C_VEL
LIN {X 0,Y 156.135,Z 747.399,A -85,B 0,C 180,E1 -25154.247,E2 -25154.247} C_VEL
